// POUs/FileHandling/TF6421-XmlServer/XmlReadWriteWithBackupFile
{attribute 'no_check'}
//Write xml files with a additonal backup file and auto save function if structure will be changed.
//For the Backup functionality, a backup subfolder name "Backup" in the directory is needed! 
//In case the xml could not read successfully after, the backup files will be used.
//See Options to enable auto save and backup file functions.
//based on TF6421 - required lib: Tc2_XmlDataSvr - see Beckhoff documentation for more information
{attribute 'enable_dynamic_creation'}
FUNCTION_BLOCK XmlReadWriteWithBackupFile EXTENDS XmlReadWrite 
VAR_OUTPUT CONSTANT
{attribute 'displaymode':='binary'}
	OPTION_ENABLE_AUTO_SAVE									:	BYTE :=2#0000_0001;
{attribute 'displaymode':='binary'}
	OPTION_ENABLE_BACKUP_FILE								: 	BYTE :=2#0000_0010;
END_VAR                 									
VAR_INPUT               									                       		
{attribute 'displaymode':='binary'}
	Options													:	BYTE := 2#0000_0000;			(* option constants are alreay predefined, so they can accordingly be passed symbolically to the block 
																								Bit 0 = Enable auto save if data changed
																								Bit 1 = Enable backup file 
																								Bit 2 = 
																								Bit 3 = 
																								Bit 4 = 
																								Bit 5 = 
																								Bit 6 = 
																								Bit 7 = 						
																							*)     													
END_VAR
VAR_OUTPUT
	Backup													:	BOOL := FALSE; 		// Backup file has been readed 
	Loaded													:	BOOL:= FALSE;		// Data loaded
	ErrorFnc												:	STRING(30) := ''; 	// Error source
END_VAR
VAR
(* memory ************************************************************)
	rtExecuteAutoSave										:	R_trig;
	pCompareData											:	POINTER TO BYTE;
	pMemSymAddr												: 	PVOID := 0;	
	MemSymSize												:	UDINT;
(* Trigger **********************************************************)

(* timer ******************************************************************)
	tonDelay												:	ton;

(* function blocks ***************************************************************)

(* Dummy **********************************************************)

END_VAR

	(* XML Read/Write with backup file and auto save						V2.2		*)
	(************************************************************************************)

(* reserver memeory for auto save ***************************************************************************************)
	IF Options.0 AND pCompareData = 0 
	THEN	
		pCompareData 										:=  __NEW(BYTE, SymSize);
		IF NOT PARAM.ENABLE_DEBUG_MSG_DYNAMIC_MEM_ALLOCATION
		THEN 
			;
		ELSIF MemSymSize = 0 
		THEN
			AdsLogHint('EngineeringToolbox | FB XmlReadWriteWithBackupFile | An instance allocated %s bytes from the dynamic memory of the ADS router memory pool', TO_STRING(SymSize));	
		ELSE //Allocation of additional memory space
			AdsLogWarn('EngineeringToolbox | FB XmlReadWriteWithBackupFile | An instance allocated additional %s bytes from the dynamic memory of the ADS router memory pool because the size of the data increased (SymSize) ', TO_STRING(SymSize));
		END_IF
		MemSymSize											:= SymSize;
	ELSIF pCompareData <> 0 
	THEN
		IF NOT Options.0 OR SymSize > MemSymSize
		THEN //Delete pointer to allocated memory if no longer needed or size increase 
			__DELETE(pCompareData);
		ELSIF pMemSymAddr <> pSymAddr OR MemSymSize <> SymSize
		THEN //Erease data and rewrite if pointer to data changed or size decreased 
			MEMSET(pCompareData,0,MemSymSize); //Delete compare data if pointer to data changed to activate auto save
			MemSymSize										:= SymSize;
			pMemSymAddr 									:= pSymAddr;	
		END_IF
	END_IF
	
(* Execute sequence ***************************************************************************)	
	rtExecuteAutoSave(CLK := Options.0 AND state = 0 AND Loaded AND pCompareData <> 0 AND_THEN MEMCMP(pSymAddr, pCompareData, SymSize) <> 0);
	rtExecute(CLK := Execute );	
	
	CASE state OF
	0:
		Busy												:= FALSE;
		// init		                                	
		IF NOT Execute                              	
		THEN                                        	
			Backup											:= FALSE;			
			Done 											:= FALSE;
			Error											:= FALSE;
			ErrorID											:= 0;
			ErrorFnc										:= '';
		END_IF                                      	
		                                            	
		IF rtExecute.Q OR rtExecuteAutoSave.Q                       	
		THEN                                        	
			Backup											:= FALSE;
			Done 											:= FALSE;
			Busy											:= TRUE;
			Error											:= FALSE;
			ErrorID											:= 0;
			ErrorFnc										:= '';
			MemFnc											:= SEL(rtExecuteAutoSave.Q, Fnc, FNC_WRITE); // write has priority
			                                        	
			IF pSymAddr = 0                         	
			THEN                                    	
				Busy										:= NOT Error;
				Error										:= TRUE;
				ErrorId										:= E_AdsErr.DEVICE_INVALIDPARM;
				Done										:= FALSE;
				MemFnc										:= -1 ;
				RETURN;                             	
			ELSE
				CASE MemFnc OF
				FNC_READ:	
					XmlSrvRead	(bExecute := FALSE,sFilePath	:= CONCAT(FilePath,FileName));
					state 									:= 10;
				FNC_WRITE:	
					XmlSrvWrite	(bExecute := FALSE,sFilePath	:= CONCAT(FilePath,FileName));
					state 									:= 20;				
				ELSE
					Error									:= TRUE;
					ErrorID									:= E_AdsErr.DEVICE_INVALIDPARM;
					ErrorFnc								:= CONCAT('Invalid Fnc,', INT_TO_STRING(MemFnc));
					Busy									:= FALSE;			
				END_CASE
			END_IF
		END_IF
	
	(* File read ************************************************)
	10:
		XmlSrvRead(                    	
			sNetId		:= NetId,
			ePath		:= ,(* Default *)
			nMode		:= XMLSRV_SKIPMISSING, 
			pSymAddr	:= pSymAddr,
			cbSymSize	:= SymSize,
			sFilePath	:= ,
			sXPath		:= XPath,
			bExecute	:=  TRUE,
			tTimeout	:= Timeout,
			bBusy		=> ,
			bError		=> ,
			nErrId		=> );
			
		IF NOT XmlSrvRead.bBusy
		THEN
			IF XmlSrvRead.bError
			THEN
				IF XmlSrvRead.nErrId = 1804 
					AND Options.1
				THEN
					state									:= 11;
				ELSE
					Error									:= TRUE;
					ErrorID									:= XmlSrvRead.nErrId;
					ErrorFnc								:= CONCAT('XmlSvrRead State:',INT_TO_STRING(State));
					Busy									:= FALSE;
					State									:= 0;	
				END_IF
			ELSE
				Loaded										:= TRUE;
				Busy										:= FALSE;
				Done										:= TRUE;
				MemFnc										:= -1;
				state										:= 0;	
				IF pCompareData <> 0 THEN MEMCPY(pCompareData,pSymAddr,SymSize); pMemSymAddr := pSymAddr; END_IF 	// refresh compare data after reading for initalisation
			END_IF
			XmlSrvRead(bExecute 							:= FALSE);
		END_IF	
				
	11: // Read Backup file
		XmlSrvRead.sFilePath								:= CONCAT(FilePath,'Backup\'); 				// subfolder
		XmlSrvRead.sFilePath								:= CONCAT(XmlSrvRead.sFilePath,FileName);
				
		XmlSrvRead(                    	
			sNetId		:= NetId,
			ePath		:= ,(* Default *)
			nMode		:= XMLSRV_SKIPMISSING, 
			pSymAddr	:= pSymAddr,
			cbSymSize	:= SymSize,
			sFilePath	:= ,
			sXPath		:= XPath,
			bExecute	:=  TRUE,
			tTimeout	:= Timeout,
			bBusy		=> ,
			bError		=> ,
			nErrId		=> );
			
		IF NOT XmlSrvRead.bBusy
		THEN
			IF XmlSrvRead.bError
			THEN
				Error										:= TRUE;
				ErrorID										:= XmlSrvRead.nErrId;
				ErrorFnc									:= CONCAT('XmlSvrRead State:',INT_TO_STRING(State));
				Busy										:= FALSE;
				State										:= 0;	
			ELSE                                        	
				Loaded										:= TRUE;
				Backup										:= TRUE;
				Busy										:= FALSE;
				Done										:= TRUE;
				MemFnc										:= -1;
				state										:= 20; 							// Write original file	
				IF pCompareData <> 0 THEN MEMCPY(pCompareData,pSymAddr,SymSize); pMemSymAddr := pSymAddr; END_IF 	// refresh compare data after reading of backup file for initalisation
			END_IF
			XmlSrvRead(bExecute 							:= FALSE);
		END_IF	
		
	(* Write parameter ***********************************************************)
	20:
		XmlSrvWrite(
			sNetId		:= NetId,
			ePath		:= ,(* Default *)
			nMode		:= Mode,
			pSymAddr	:= pSymAddr,
			cbSymSize	:= SymSize,
			sFilePath	:= ,
			sXPath		:= XPath,
			bExecute	:= TRUE,
			tTimeout	:= Timeout,
			bBusy		=> ,
			bError		=> ,
			nErrId		=> );
			
		IF NOT XmlSrvWrite.bBusy
		THEN
			IF XmlSrvWrite.bError
			THEN
				Error										:= TRUE;
				ErrorID										:= XmlSrvWrite.nErrId;
				ErrorFnc									:= CONCAT('XmlSvrWrite State:',INT_TO_STRING(State));
				Busy										:= FALSE;
				State										:= 0;				
			ELSE // Write backup file	
				Loaded										:= TRUE;
				State										:= SEL(Options.1, 0, 21); //
				Done										:= State = 0; 				
				Busy										:= State <> 0;
				//Update compare memory
				IF pCompareData <> 0 THEN MEMCPY(pCompareData,pSymAddr,SymSize); pMemSymAddr := pSymAddr; END_IF 	// refresh compare data after writing new data
			END_IF
			XmlSrvWrite(bExecute							:= FALSE);
		END_IF

	21://Write backup to sub folder	
		XmlSrvWrite.sFilePath								:= CONCAT(FilePath,'Backup\'); 				// subfolder
		XmlSrvWrite.sFilePath								:= CONCAT(XmlSrvWrite.sFilePath,FileName);
		XmlSrvWrite(
			sNetId		:= NetId,
			ePath		:= ,(* Default *)
			nMode		:= Mode,
			pSymAddr	:= pSymAddr,
			cbSymSize	:= SymSize,
			sFilePath	:= ,
			sXPath		:= XPath,
			bExecute	:= TRUE,
			tTimeout	:= Timeout,
			bBusy		=> ,
			bError		=> ,
			nErrId		=> );
			
		IF NOT XmlSrvWrite.bBusy
		THEN
			IF XmlSrvWrite.bError
			THEN
				Error										:= TRUE;
				ErrorID										:= XmlSrvWrite.nErrId;
				ErrorFnc									:= CONCAT('XmlSvrWrite State:',INT_TO_STRING(State));
				Busy										:= FALSE;
				State										:= 0;				
			ELSE 	
				Busy										:= FALSE;
				Done										:= TRUE;
				State										:= 0;	
				//Update compare memory
				IF pCompareData <> 0 THEN MEMCPY(pCompareData,pSymAddr,SymSize); pMemSymAddr := pSymAddr; END_IF 	// refresh compare data after writing new data				
			END_IF
			XmlSrvWrite(bExecute							:= FALSE);
		END_IF		
	END_CASE
		
		
	
(*************************************************************************************************)

METHOD FB_exit : BOOL
VAR_INPUT
	bInCopyCode : BOOL; // if TRUE, the exit method is called for exiting an instance that is copied afterwards (online change).
END_VAR
IF NOT bInCopyCode AND pCompareData <> 0
THEN //Release memory in case the PLC stopps
	__DELETE(pCompareData);
END_IF
END_METHOD

PROPERTY PUBLIC optEnableAutoSave : BOOL
GET
optEnableAutoSave := Options.0;
END_GET
SET
Options.0 := optEnableAutoSave;
END_SET
END_PROPERTY

PROPERTY PUBLIC optEnableBackupFile : BOOL
GET
optEnableBackupFile := Options.1;
END_GET
SET
Options.1 := optEnableBackupFile;
END_SET
END_PROPERTY

METHOD PUBLIC read : BOOL //Return value = TRUE if busy
//required parameter
//pSymAddr
//SymSize
//FilePath
//XPath
VAR_INPUT
	Execute													:	BOOL;
END_VAR
CASE state OF
0:	
	Fnc 													:= FNC_READ;
	THIS^(Execute:=Execute);
1: 
	;

END_CASE
Read 														:= Busy;
END_METHOD

METHOD PUBLIC write : BOOL //Return value = TRUE if busy
//required parameter
//pSymAddr
//SymSize
//FilePath
//XPath
VAR_INPUT
	Execute													:	BOOL;
END_VAR
CASE state OF
0:	
	Fnc 													:= FNC_WRITE;
	THIS^(Execute:=Execute);
1: 
	;

END_CASE
Write 														:= Busy;
END_METHOD

END_FUNCTION_BLOCK

// POUs/IO/_EcSlaveFWUpdater/EcSlaveDevFWUpdater
FUNCTION_BLOCK EcSlaveDevFWUpdater EXTENDS FbBase
VAR CONSTANT	
	{attribute 'displaymode':='hexadecimal'} 
	COE_FWVERSION_OBJECT								: WORD := 16#100A;
END_VAR
VAR_OUTPUT CONSTANT
	MIN_SLAVE_DEV										:	INT := 1;
	MAX_SLAVE_DEV										:	INT := Param.ETHERCAT_SLAVE_DEV_FW_UPDATER_MAX_DEV;

	{attribute 'displaymode':='binary'}   
	MODE_READ											:	BYTE := 0;
	{attribute 'displaymode':='binary'}   
	MODE_WRITE											:	BYTE := 1;

	{attribute 'displaymode':='binary'}   
	OPTION_WRITE_FW_IF_VERSION_MATCH					:	BYTE := 2#0000_0001;
	
END_VAR
VAR_INPUT
{attribute 'displaymode':='binary'}         			
	Mode												:	BYTE  := 2#0000_0000; 

{attribute 'displaymode':='binary'}  	
	Options												:	BYTE  := 2#0000_0000; 		
				
	PathName											:	STRING; //Path incl. file name of FW file
	RegVersion											:	STRING; //Requested version
	ipSlaveInfoData										:	ARRAY [MIN_SLAVE_DEV..MAX_SLAVE_DEV] OF I_EcSlaveInfoData;
END_VAR
VAR_OUTPUT
	ActVersion											: ARRAY[MIN_SLAVE_DEV..MAX_SLAVE_DEV] OF STRING[20]; 	
	CntFWNOK											: INT; //Count of terminals FW not OK
	TermNo												: INT; //No of terminal in progress
	ProgressWriteFW										: UDINT;	
	VersionRead											: BOOL;
END_VAR
VAR
(*  Memory *****************************************************)
	lastState											: INT := 0;
	MinTerm												: INT;

(*  Timer ******************************************************)
(*  Trigger ****************************************************)

(*  Blocks *****************************************************)
	EcCoeSdoReadEx										: FB_EcCoeSdoReadEx := (nIndex := COE_FWVERSION_OBJECT, tTimeout := DEFAULT_ADS_TIMEOUT);

	CoEFwDownLoad										: FB_EcFoeLoad := (tTimeout := DEFAULT_ADS_TIMEOUT,dwPass := 0, eMode := eFoeMode_Write);
(*  Error ******************************************************)
(*  Dummys *****************************************************)
	{attribute 'hide' := ''}
	i,j													: INT := 0;

END_VAR

	(*********************************************************)
	
(* state machine ********************************************************)
	rtExecute(CLK := Execute);
	CASE state OF
	0 : 
		Busy 											:= FALSE;
		
		IF NOT Execute THEN
			Done 										:= FALSE;
			Error 										:= FALSE;
			ErrorID 									:= 0;
		END_IF
		IF rtExecute.Q THEN
			IF PathName = '' 
			THEN
				Error 									:= TRUE;
				ErrorID 								:= E_AdsErr.DEVICE_INVALIDPARM;

			ELSIF RegVersion = '' AND Mode = MODE_WRITE AND NOT Options.0
			THEN
 				Error 									:= TRUE;
				ErrorID 								:= E_AdsErr.DEVICE_INVALIDPARM; 
									
			ELSIF ipSlaveInfoData[MIN_SLAVE_DEV] = 0
			THEN
 				Error 									:= TRUE;
				ErrorID 								:= E_AdsErr.DEVICE_INVALIDPARM; 			
			ELSE
				Busy									:= TRUE;	
				Done 									:= FALSE;
				Error 									:= FALSE;
				ErrorID 								:= 0;
				TermNo									:= MIN_SLAVE_DEV;	
				ProgressWriteFW							:= 0;
				CntFWNOK								:= 0;					
				
			
				EcCoeSdoReadEx(bExecute := FALSE);
				CoEFwDownLoad(bExecute := FALSE);
				state									:= SEL(Mode = MODE_READ, 1, 2);
			END_IF
		END_IF
			
	1: (* Write FW *****************************************************************)
		CoEFwDownLoad(
			bExecute		:= ipSlaveInfoData[TermNo].rInfoData.AdsAddr.port <> 0 AND (ActVersion[TermNo] <> RegVersion OR Options.0) , 
			sNetId			:= F_CreateAmsNetId(nIds := ipSlaveInfoData[TermNo].rInfoData.AdsAddr.netId),
			nSlaveAddr		:= ipSlaveInfoData[TermNo].rInfoData.AdsAddr.port,
			sPathName		:= PathName,
			nProgress 		=> ProgressWriteFW);	
		IF NOT 	CoEFwDownLoad.bBusy
		THEN
			ProgressWriteFW								:= 0;
			IF CoEFwDownLoad.bError
			THEN
				ErrorID									:= EcCoESdoReadEx.nErrId;
				CntFWNOK								:= CntFWNOK + 1;	
				ActVersion[TermNo]						:= 'ERR_DOWNLOADING';
			ELSIF CoEFwDownLoad.bExecute	
			THEN
				ActVersion[TermNo]						:= 'DOWNLOADED';
			ELSE
				ActVersion[TermNo]						:= '------';
			END_IF
			//Next terminal
			TermNo										:= TermNo + 1;
			
			IF TermNo > MAX_SLAVE_DEV 
				OR ipSlaveInfoData[TermNo] = 0
			THEN //Start reading
				MEMSET(ADR(ActVersion),0,SIZEOF(ActVersion));
				VersionRead								:= FALSE;
				TermNo									:= MIN_SLAVE_DEV;		
				state									:= 2;
			END_IF		
			CoEFwDownLoad(bExecute := FALSE);
		ELSE
			ActVersion[TermNo]							:= CONCAT('DOWNLOADING ',CONCAT(TO_STRING(CoEFwDownLoad.nProgress),'%'));
		END_IF
	
	2: (* Read FW Version **********************************************************)
		EcCoESdoReadEx(
			bExecute		:= ipSlaveInfoData[TermNo].rInfoData.AdsAddr.port <> 0,
			sNetId			:= F_CreateAmsNetId(nIds := ipSlaveInfoData[TermNo].rInfoData.AdsAddr.netId),
			nSlaveAddr		:= ipSlaveInfoData[TermNo].rInfoData.AdsAddr.port,
			pDstBuf			:= ADR(ActVersion[TermNo]),
			cbBufLen		:= SIZEOF(ActVersion[TermNo]));
		IF NOT EcCoESdoReadEx.bBusy
		THEN
			IF EcCoESdoReadEx.bError 
			THEN
				ActVersion[TermNo]						:= 'ERR_READING';
				ErrorID									:= EcCoESdoReadEx.nErrId;
				CntFWNOK								:= CntFWNOK + 1;	
			ELSIF NOT EcCoESdoReadEx.bExecute 
			THEN
				ActVersion[TermNo]						:= 'NOT_CONNECTED';
			ELSIF ActVersion[TermNo] <> RegVersion
			THEN
				CntFWNOK								:= CntFWNOK + 1;	
			END_IF
			
			//Next terminal
			TermNo										:= TermNo + 1;
			
			IF TermNo > MAX_SLAVE_DEV
				OR ipSlaveInfoData[TermNo] = 0
			THEN
				TermNo									:= MAX_SLAVE_DEV;
				Done									:= CntFWNOK = 0;
				VersionRead								:= TRUE;
				Error									:= NOT Done;
				Busy									:= FALSE;
				state									:= 0;
			END_IF
			EcCoeSdoReadEx(bExecute := FALSE);
		END_IF
	END_CASE	

(* Record last state ******************************************)
IF state <> lastState AND state <> 0 AND NOT Error
THEN 
	lastState											:= state;
END_IF

(*************************************************************)

END_FUNCTION_BLOCK

// POUs/IO/_ItfActuators/I_ActuatorBase
INTERFACE I_ActuatorBase EXTENDS __System.IQueryInterface

{attribute 'monitoring' := 'call'}
PROPERTY public inError : bool
GET
END_GET
END_PROPERTY

{attribute 'monitoring' := 'call'}
PROPERTY public isBusy : bool
GET
END_GET
END_PROPERTY

{attribute 'monitoring' := 'call'}
PROPERTY public isOff : BOOL
GET
END_GET
END_PROPERTY

{attribute 'monitoring' := 'call'}
PROPERTY public noFeed : BOOL
GET
END_GET
END_PROPERTY

{attribute 'monitoring' := 'call'}
PROPERTY public ok : bool
GET
END_GET
END_PROPERTY

METHOD PUBLIC reset : BOOL
VAR_INPUT
END_VAR
END_METHOD

METHOD public switchOff : BOOL
VAR_INPUT
END_VAR
END_METHOD

END_INTERFACE

// POUs/IO/_ItfActuators/I_ActuatorEnableDisable
INTERFACE I_ActuatorEnableDisable EXTENDS I_ActuatorBase

{attribute 'monitoring' := 'call'}
PROPERTY public isDisabled : BOOL
GET
END_GET
END_PROPERTY

{attribute 'monitoring' := 'call'}
PROPERTY public isEnabled : BOOL
GET
END_GET
END_PROPERTY

METHOD public setDisable : BOOL
VAR_INPUT
END_VAR
END_METHOD

METHOD public setEnable : BOOL
VAR_INPUT
END_VAR
END_METHOD

END_INTERFACE

// POUs/IO/_ItfActuators/I_ActuatorFwdBwd
INTERFACE I_ActuatorFwdBwd EXTENDS I_ActuatorBase

{attribute 'monitoring' := 'call'}
PROPERTY public backwardStarted : BOOL
GET
END_GET
END_PROPERTY

{attribute 'monitoring' := 'call'}
PROPERTY public forwardStarted : BOOL
GET
END_GET
END_PROPERTY

METHOD public startBackward : BOOL
VAR_INPUT
END_VAR
END_METHOD

METHOD public startForward : BOOL
VAR_INPUT
END_VAR
END_METHOD

END_INTERFACE

// POUs/IO/_ItfActuators/I_ActuatorFwdRev
INTERFACE I_ActuatorFwdRev EXTENDS I_ActuatorBase

{attribute 'monitoring' := 'call'}
PROPERTY public forwardStarted : BOOL
GET
END_GET
END_PROPERTY

{attribute 'monitoring' := 'call'}
PROPERTY public reverseStarted : BOOL
GET
END_GET
END_PROPERTY

METHOD public startForward : BOOL
VAR_INPUT
END_VAR
END_METHOD

METHOD public startReverse : BOOL
VAR_INPUT
END_VAR
END_METHOD

END_INTERFACE

// POUs/IO/_ItfActuators/I_ActuatorLeftRight
INTERFACE I_ActuatorLeftRight EXTENDS I_ActuatorBase

{attribute 'monitoring' := 'call'}
PROPERTY public leftOk : BOOL
GET
END_GET
END_PROPERTY

{attribute 'monitoring' := 'call'}
PROPERTY public rightOk : BOOL
GET
END_GET
END_PROPERTY

METHOD public toTheLeft : BOOL
VAR_INPUT
END_VAR
END_METHOD

METHOD public toTheRight : BOOL
VAR_INPUT
END_VAR
END_METHOD

END_INTERFACE

// POUs/IO/_ItfActuators/I_ActuatorOnOff
INTERFACE I_ActuatorOnOff EXTENDS I_ActuatorBase

{attribute 'monitoring' := 'call'}
PROPERTY public isOn : BOOL
GET
END_GET
END_PROPERTY

METHOD public switchOn : BOOL
VAR_INPUT
END_VAR
END_METHOD

END_INTERFACE

// POUs/IO/_ItfActuators/I_ActuatorOpenClose
INTERFACE I_ActuatorOpenClose EXTENDS I_ActuatorBase

{attribute 'monitoring' := 'call'}
PROPERTY public isClosed : BOOL
GET
END_GET
END_PROPERTY

{attribute 'monitoring' := 'call'}
PROPERTY public isOpened : BOOL
GET
END_GET
END_PROPERTY

METHOD public setClose : BOOL
VAR_INPUT
END_VAR
END_METHOD

METHOD public setOpen : BOOL
VAR_INPUT
END_VAR
END_METHOD

END_INTERFACE

// POUs/IO/_ItfActuators/I_ActuatorPosNeg
INTERFACE I_ActuatorPosNeg EXTENDS I_ActuatorBase

{attribute 'monitoring' := 'call'}
PROPERTY public negativeOk : BOOL
GET
END_GET
END_PROPERTY

METHOD PUBLIC negativeOn : BOOL
VAR_INPUT
END_VAR
END_METHOD

{attribute 'monitoring' := 'call'}
PROPERTY public positiveOk : BOOL
GET
END_GET
END_PROPERTY

METHOD PUBLIC positiveOn : BOOL
VAR_INPUT
END_VAR
END_METHOD

END_INTERFACE

// POUs/IO/_ItfActuators/I_ActuatorStartStop
INTERFACE I_ActuatorStartStop EXTENDS I_ActuatorBase

{attribute 'monitoring' := 'call'}
PROPERTY public isStarted : BOOL
GET
END_GET
END_PROPERTY

{attribute 'monitoring' := 'call'}
PROPERTY public isStopped : BOOL
GET
END_GET
END_PROPERTY

METHOD public start : BOOL
VAR_INPUT
END_VAR
END_METHOD

METHOD public stop : BOOL
VAR_INPUT
END_VAR
END_METHOD

END_INTERFACE

// POUs/IO/_ItfActuators/I_ActuatorUpDown
INTERFACE I_ActuatorUpDown EXTENDS I_ActuatorBase

{attribute 'monitoring' := 'call'}
PROPERTY public downOk : BOOL
GET
END_GET
END_PROPERTY

METHOD public moveDown : BOOL
VAR_INPUT
END_VAR
END_METHOD

METHOD public moveUp : BOOL
VAR_INPUT
END_VAR
END_METHOD

{attribute 'monitoring' := 'call'}
PROPERTY public upOK : BOOL
GET
END_GET
END_PROPERTY

END_INTERFACE

// POUs/IO/_ItfActuators/I_ActuatorWorkBase
INTERFACE I_ActuatorWorkBase EXTENDS I_ActuatorBase

{attribute 'monitoring' := 'call'}
PROPERTY isInBasePos : BOOL
GET
END_GET
END_PROPERTY

{attribute 'monitoring' := 'call'}
PROPERTY isInWorkPos : BOOL
GET
END_GET
END_PROPERTY

METHOD public moveToBasePos : BOOL
VAR_INPUT
END_VAR
END_METHOD

METHOD public moveToWorkPos : BOOL
VAR_INPUT
END_VAR
END_METHOD

END_INTERFACE

// POUs/IO/Analog/AnalogIn32
{attribute 'no_check'}
FUNCTION_BLOCK AnalogIn32 extends EcSlaveInfoDataExt
VAR_INPUT
	MinValue												: 	LREAL 	:= 0.0;
	MaxValue												: 	LREAL 	:= 0.0;
	NoOfDigits												: 	INT 	(0..10)	:= 0; //number of decimal digits of scaled Q variable 
	OutOnError												:	LREAL 	:= 0.000000000000000001;
{attribute 'displaymode':='binary'}     	            	
	Options													:	BYTE  := 2#0000_0010; (* .0 = FALSE Scale value from 0 to e.g. 32767 / TRUE scale singed value e.g. -32768 <-> 32767 , see Options .1 and .2 for more scaling Options 
																						.1 = FALSE = 32 bit resolution / TRUE = value is based on 24 bit resolution e.g. -> -8388608.0 or 0.0 <-> 8388607.0 
																						.2 = Right adjust of 32/24 bit value -> value will be shifted by 8 bits (divided bv 256)   
																						.3 = TRUE = Enable extended range mode -> change scaling to +/-7812500 instead of r+/- 838860x *)
	Offset													:	LREAL := 0.0;
END_VAR                 									                                	            	
VAR_OUTPUT                              	            	
	Q														:	LREAL;	//scaled result value
	In											AT  %I* 	: 	DINT; 	//Hardware Input 
{attribute 'displaymode':='binary'}     	            	
	Status										AT  %I*		:	WORD := 2#0100_0000_0000_0000;	//Terminal status word -> can also be linked with status byte
END_VAR

(* read 32bit analog value 																				    *)
(* resolution process image			e.g.				/ 0V = 0 / 10V = 2147483647 / -10V = - 2147483647 	*)
(* or directly with NoOfDigits																	250 -> 25.0°*)
(************************************************************************************************************)
	
(* Scaling ******************************************************************)
	IF MaxValue <> MinValue 
	THEN
		IF Options.1 
		THEN //24 bit resolution
			IF NOT Options.3
			THEN
				Q 	 										:= Offset + scale(SEL(Options.2 , In , In / 256.0 ) , SEL(Options.0, 0.0, -8388608.0), 8388607.0, MinValue , MaxValue);
			ELSE
		 		Q 	 										:= Offset + scale(SEL(Options.2 , In , In / 256.0 ) , SEL(Options.0, 0.0, -7812500.0), 7812500.0, MinValue , MaxValue);
			END_IF
		ELSE //32 bit resolution 
			Q 	 											:= Offset + scale(SEL(Options.2 , In , In / 256.0 ) , SEL(Options.0, 0.0, -2147483648.0), 2147483647.0, MinValue , MaxValue);		
		END_IF
		IF NoOfDigits > 0
		THEN
			Q												:= TO_FMLREAL(Q,NoOfDigits);
		END_IF
	
	ELSIF NoOfDigits > 0 (* Bsp PT100 *)
	THEN
		Q													:= Offset + TO_FMLREAL(In,NoOfDigits);
		
	ELSE  													
		Q 													:= 0.0;
	END_IF

	IF 	Error AND OutOnError <> 0.000000000000000001
	THEN
		Q													:= OutOnError;
	END_IF
(**********************************************************************************************************************)

{attribute 'monitoring' := 'call'}
PROPERTY PUBLIC Error : BOOL
GET
Error					:= Status.6 OR MinValue = MaxValue AND NoOfDigits = 0;
END_GET
END_PROPERTY

{attribute 'monitoring' := 'call'}
PROPERTY PUBLIC Limit_1 : BYTE
GET
Limit_1.0					:= Status.2;
Limit_1.1					:= Status.3;
END_GET
END_PROPERTY

{attribute 'monitoring' := 'call'}
PROPERTY PUBLIC Limit_2 : BYTE
GET
Limit_2.0					:= Status.4;
Limit_2.1					:= Status.5;
END_GET
END_PROPERTY

PROPERTY optEnable24BitResolution : BOOL //In value is provided as 32bit value instead if 24bit
GET
optEnable24BitResolution := Options.1;
END_GET
SET
Options.1 := optEnable24BitResolution;
END_SET
END_PROPERTY

PROPERTY PUBLIC optEnableScaleExtRangeMode : bool
GET
optEnableScaleExtRangeMode := Options.3;
END_GET
SET
Options.3 := optEnableScaleExtRangeMode;
END_SET
END_PROPERTY

PROPERTY PUBLIC optEnableScaleSignedValue : bool
GET
optEnableScaleSignedValue := Options.0;
END_GET
SET
Options.0 := optEnableScaleSignedValue;
END_SET
END_PROPERTY

PROPERTY PUBLIC optShiftValueBy8Bits : BOOL
GET
optShiftValueBy8Bits := Options.2;
END_GET
SET
Options.2 := optShiftValueBy8Bits;
END_SET
END_PROPERTY

{attribute 'monitoring' := 'call'}
PROPERTY PUBLIC Overrange : BOOL
GET
Overrange					:= Status.1;
END_GET
END_PROPERTY

{attribute 'monitoring' := 'call'}
PROPERTY PUBLIC SyncError : BOOL
GET
SyncError 			:= Status.13;
END_GET
END_PROPERTY

{attribute 'monitoring' := 'call'}
PROPERTY PUBLIC TxPDOState : BOOL
GET
TxPDOState					:= Status.14; //True if not valid
END_GET
END_PROPERTY

{attribute 'monitoring' := 'call'}
PROPERTY PUBLIC TxPDOToggle : BOOL
GET
TxPDOToggle						:= Status.15;
END_GET
END_PROPERTY

{attribute 'monitoring' := 'call'}
PROPERTY PUBLIC Underrange : BOOL
GET
Underrange 					:= Status.0;
END_GET
END_PROPERTY

END_FUNCTION_BLOCK

// POUs/IO/Analog/AnalogInELMBase
// Based FB for analog input channels of ELM terminals incl. EtherCAT Slave Info Data 
//You can inherit your final implementation from this base "class"  
FUNCTION_BLOCK AnalogInELMBase EXTENDS EcSlaveInfoData
VAR_INPUT
	Enable													:	BOOL 	:= TRUE;
	MinValue												: 	LREAL 	:= 0.0;
	MaxValue												: 	LREAL 	:= 0.0;
	NoOfDigits												: 	INT 	(0..10)	:= 0; //number of decimal digits of scaled Q variable 
	OutOnError												:	LREAL 	:= 0.000000000000000001;
{attribute 'displaymode':='binary'}     	            	
	Options													:	BYTE  := 2#0000_0000;
END_VAR                 									
VAR                                     	            	
{attribute 'displaymode':='binary'}     	            	
	Status										AT  %I*		:	DWORD := 2#0100_0000_0000_0000;	//Terminal status (4 bytes) 
	
END_VAR                                 	            	
VAR_OUTPUT                              	            	                                       	
	(* Statusbist *)                    	
	NoOfSamples												:	USINT; //Byte 1
	Error													:	BOOL; //Byte2.0
	Underrange 												:	BOOL; //Byte2.1
	Overrange												:	BOOL ; //Byte2.2
	Diag													:	BOOL; //Byte2.4
	TxPDOState												:	BOOL; //Byte2.5
	InputCycleCounter										:	USINT; //Byte2.6/.7	
END_VAR                                 	
VAR                                     	
END_VAR

(* Base FB for ELM analog in terminals 																		*)
(************************************************************************************************************)

(* evaluate statusword **************************************************************************************)
	MEMCPY(ADR(NoOfSamples),ADR(Status),SIZEOF(NoOfSamples));
	Error													:= Enable AND (Status.8 OR MinValue = MaxValue AND NoOfDigits = 0);
	Underrange 												:= Status.9;
	Overrange												:= Status.10;
	
	Diag													:= Status.12;
	TxPDOState												:= Status.13; //True if not valid
	InputCycleCounter.0										:= Status.14;
	InputCycleCounter.1										:= Status.15;
	
(**********************************************************************************************************************)

END_FUNCTION_BLOCK

// POUs/IO/Analog/AnalogInELMSingleSampleDINT
// AnalogIn FB to read and scale a single DINT (24bit) sample input from ELMxxxx terminal
// Set bit 3 (Options.3) to true to enable scaling based on +/-7812500 instead of legacy range values +/-838860x
FUNCTION_BLOCK AnalogInELMSingleSampleDINT EXTENDS AnalogInELMBase
VAR_INPUT
	Offset													:	LREAL := 0.0;

END_VAR                 									
VAR                                     	            	
END_VAR                                 	            	
VAR_OUTPUT                              	            	                                       	
	Q														:	LREAL;	//scaled result value
	In											AT  %I* 	: 	DINT; 	//Hardware Input 
END_VAR                                 	
VAR                                   	
END_VAR

(* Read single DINT sample value from ELM terminal and scale to user units									*)
(************************************************************************************************************)

(* evaluate statusword **************************************************************************************)
	SUPER^();
	
(* Scaling ******************************************************************)
	IF MaxValue <> MinValue 
	THEN	
		IF NOT Options.3
		THEN
			Q 	 											:= Offset + Scale(TO_LREAL(In) , -8388608.0, 8388607.0, MinValue , MaxValue);
		ELSE
			Q 	 											:= Offset + Scale(TO_LREAL(In), -7812500.0, 7812500.0, MinValue , MaxValue);
		END_IF	
		IF NoOfDigits > 0
		THEN
			Q												:= TO_FMLREAL(Q,NoOfDigits);
		END_IF
	
	ELSIF NoOfDigits > 0 (* Bsp PT100 *)
	THEN
		Q													:= Offset + TO_FMLREAL(In,NoOfDigits);
		
	ELSE  													
		Q 													:= 0.0;
	END_IF

	IF 	Error AND OutOnError <> 0.000000000000000001
	THEN
		Q													:= OutOnError;
	END_IF
(**********************************************************************************************************************)

METHOD FB_init : BOOL
VAR_INPUT
	bInitRetains : BOOL; // if TRUE, the retain variables are initialized (warm start / cold start)
	bInCopyCode : BOOL;  // if TRUE, the instance afterwards gets moved into the copy code (online change)
END_VAR
IF NOT bInCopyCode THEN
	NoOfDigits 							:= 2;
END_IF
END_METHOD

PROPERTY PUBLIC optEnableScaleExtRangeMode : bool
GET
optEnableScaleExtRangeMode := Options.3;
END_GET
SET
Options.3 := optEnableScaleExtRangeMode;
END_SET
END_PROPERTY

END_FUNCTION_BLOCK

// POUs/IO/Analog/AnalogInELMSingleSampleREAL
// AnalogIn FB to read and scale a single REAL sample input from ELMxxxx terminal
// Set bit 3 (Options.3) to true to enable scaling based on +/-7812500 instead of legacy range values +/-838860x
// NoOfDigits per default set to 3... 
FUNCTION_BLOCK AnalogInELMSingleSampleREAL EXTENDS AnalogInELMBase
VAR_INPUT
	Offset													:	LREAL := 0.0;
END_VAR                 									
VAR                                     	            	
END_VAR                                 	            	
VAR_OUTPUT                              	            	                                       	
	Q														:	LREAL;	//scaled result value
	In											AT  %I* 	: 	REAL; 	//Hardware Input 
END_VAR                                 	
VAR                                     	
END_VAR

(* Read single REAL sample value from ELM terminal and scale to user units									*)
(************************************************************************************************************)

(* evaluate statusword **************************************************************************************)
	SUPER^();
	
(* Scaling ******************************************************************)
	IF MaxValue <> MinValue 
	THEN			
		IF NOT Options.3
		THEN
			Q 	 											:= Offset + Scale(TO_LREAL(In), -8388608.0, 8388607.0, MinValue , MaxValue);
		ELSE
			Q 	 											:= Offset + Scale(TO_LREAL(In),  -7812500.0, 7812500.0, MinValue , MaxValue);		
		END_IF	
		
		IF NoOfDigits > 0
		THEN
			Q												:= TO_FMLREAL(Q,NoOfDigits);
		END_IF
	
	ELSIF NoOfDigits > 0 (* Bsp PT100 *)
	THEN
		Q													:= Offset + TO_FMLREAL(In,NoOfDigits);
		
	ELSE  													
		Q 													:= 0.0;
	END_IF


(**********************************************************************************************************************)

METHOD FB_init : BOOL
VAR_INPUT
	bInitRetains : BOOL; // if TRUE, the retain variables are initialized (warm start / cold start)
	bInCopyCode : BOOL;  // if TRUE, the instance afterwards gets moved into the copy code (online change)
END_VAR
IF NOT bInCopyCode THEN
	NoOfDigits 							:= 3;
END_IF
END_METHOD

PROPERTY PUBLIC optEnableScaleExtRangeMode : bool
GET
optEnableScaleExtRangeMode := Options.3;
END_GET
SET
Options.3 := optEnableScaleExtRangeMode;
END_SET
END_PROPERTY

END_FUNCTION_BLOCK

// POUs/IO/Analog/AnalogInREAL
// AnalogInReal FB to read and scale a single REAL input
// Set bit 3 (Options.3) to true to enable scaling based on +/-7812500 instead of legacy range values +/-838860x
// NoOfDigits per default set to 3... 
FUNCTION_BLOCK AnalogInREAL EXTENDS EcSlaveInfoDataExt
VAR_INPUT
	Offset													:	LREAL 		:= 0.0;
	MinValue												: 	LREAL 		:= 0.0;
	MaxValue												: 	LREAL 		:= 0.0;
	NoOfDigits												: 	INT(0..10)	:= 0; //number of decimal digits of scaled Q variable 
	OutOnError												:	LREAL 		:= 0.000000000000000001;
{attribute 'displaymode':='binary'}     	            	
	Options													:	BYTE  		:= 2#0000_0000;
END_VAR                 									
VAR                        
END_VAR                                 	            	
VAR_OUTPUT                              	            	                                       	
	Q														:	LREAL;//scaled result value
	In											AT  %I* 	: 	REAL; //Hardware Input
	{attribute 'displaymode':='binary'}     	            	
	Status										AT  %I*		:	WORD := 2#00000000_00000000;	//Terminal status (2 bytes)
END_VAR

(* Read single REAL value from terminal and scale to user units				*)
(****************************************************************************)

(* Scaling ******************************************************************)
	IF MaxValue <> MinValue 
	THEN			
		IF NOT Options.3
		THEN
			Q 	 											:= Offset + Scale(TO_LREAL(In), -8388608.0, 8388607.0, MinValue , MaxValue);
		ELSE
			Q 	 											:= Offset + Scale(TO_LREAL(In),  -7812500.0, 7812500.0, MinValue , MaxValue);		
		END_IF	
		
		IF NoOfDigits > 0
		THEN
			Q												:= TO_FMLREAL(Q,NoOfDigits);
		END_IF
	
	ELSIF NoOfDigits > 0 (* Bsp PT100 *)
	THEN
		Q													:= Offset + TO_FMLREAL(In,NoOfDigits);
		
	ELSE  													
		Q 													:= 0.0;
	END_IF

(****************************************************************************)

{attribute 'monitoring' := 'call'}
PROPERTY PUBLIC Error : BOOL
GET
Error					:= Status.6 OR MinValue = MaxValue AND NoOfDigits = 0;
END_GET
END_PROPERTY

{attribute 'monitoring' := 'call'}
PROPERTY PUBLIC Limit_1 : BYTE
GET
Limit_1.0					:= Status.2;
Limit_1.1					:= Status.3;
END_GET
END_PROPERTY

{attribute 'monitoring' := 'call'}
PROPERTY PUBLIC Limit_2 : BYTE
GET
Limit_2.0					:= Status.4;
Limit_2.1					:= Status.5;
END_GET
END_PROPERTY

PROPERTY PUBLIC optEnableScaleExtRangeMode : bool
GET
optEnableScaleExtRangeMode := Options.3;
END_GET
SET
Options.3 := optEnableScaleExtRangeMode;
END_SET
END_PROPERTY

{attribute 'monitoring' := 'call'}
PROPERTY PUBLIC Overrange : BOOL
GET
Overrange 			:= Status.1;
END_GET
END_PROPERTY

{attribute 'monitoring' := 'call'}
PROPERTY PUBLIC TareActive : BOOL
GET
TareActive					:= Status.11;
END_GET
END_PROPERTY

{attribute 'monitoring' := 'call'}
PROPERTY PUBLIC TxPDOState : BOOL
GET
TxPDOState					:= Status.14; //True if not valid
END_GET
END_PROPERTY

{attribute 'monitoring' := 'call'}
PROPERTY PUBLIC TxPDOToggle : BOOL
GET
TxPDOToggle							:= Status.15;
END_GET
END_PROPERTY

{attribute 'monitoring' := 'call'}
PROPERTY PUBLIC Underrange : BOOL
GET
Underrange 			:= Status.0;
END_GET
END_PROPERTY

END_FUNCTION_BLOCK

// POUs/IO/Analog/AnalogOut
{attribute 'no_check'}
//Provides an INT output varibale (Q	AT  %Q* : 	INT) to writed a scaled lreal value to an anallog output (terminal)
FUNCTION_BLOCK AnalogOut
VAR_INPUT
	SetValue												: 	LREAL 	:= 0.0;	
	MinValue												: 	LREAL 	:= 0.0;
	MaxValue												: 	LREAL 	:= 0.0;	
{attribute 'displaymode':='binary'}
	Options													:	BYTE 	:= 2#0000_0000; (* .0 = FALSE scale output to 0 - 32767 / TRUE = scale output from -32768 to +32767 *)
END_VAR             							
VAR_OUTPUT          							
	Q												AT  %Q* : 	INT; (* Hardware Output *)
END_VAR             							
VAR                 							
	x														:	LREAL;
END_VAR

(* Analogvalue output	 													    *)
(* resolution  							/ 0V = 0 / 10V = 32768 / -10V = - 32767 *)
(********************************************************************************)

(* standardization **************************************************************)
	Q															:= TO_INT(Scale(SetValue,MinValue,MAxValue,SEL(Options.0 , 0.0  , -32768.0), 32767.0));		

(*********************************************************************************)

PROPERTY PUBLIC optEnableScaleSignedValue : bool
GET
optEnableScaleSignedValue := Options.0;
END_GET
SET
Options.0 := optEnableScaleSignedValue;
END_SET
END_PROPERTY

END_FUNCTION_BLOCK

// POUs/IO/Cylinder/Cylinder
{attribute 'no_check'}
//Cylinder object with two outputs (Workpos./Basepos) and correlated inputs
//Via the Options byte, it is possible to disable the use either of one or both feedback inputs.
//In case the physical feedback input in disabled, the status output of the FB will be generated by PT_Feedback
//In case the physical feedback input will not be triggerd to his corresonding outout within a certain time (PT_Feedback), an timeout error occures
//The physical outputs could be blocked by set the FeedxxxPos signals to false.
//FB "INPUT" is used inside
FUNCTION_BLOCK Cylinder IMPLEMENTS I_Cylinder
VAR_OUTPUT CONSTANT
{attribute 'displaymode':='binary'}
	OPTION_DISABLE_SENSOR_BASEPOS							:	BYTE  := 2#0000_0001; //Disable sensor check basepos. Feedback time used instead to create signal
{attribute 'displaymode':='binary'}
	OPTION_DISABLE_SENSOR_WORKPOS							:	BYTE  := 2#0000_0010; //Disable sensor check workpos. Feedback time used instead to create signal
{attribute 'displaymode':='binary'}
	OPTION_FREE												:	BYTE  := 2#0000_0100; //Not used option		
{attribute 'displaymode':='binary'}
	OPTION_DISABLE_LOGIC_ERROR								:	BYTE  := 2#0000_1000; //Disable logic error (Sensor workpos and basepos active at the same time) 	
{attribute 'displaymode':='binary'}
	OPTION_SWAP_SENSOR_STATUS								:	BYTE  := 2#0001_0000; //Swap signals work and base pos at Status byte
{attribute 'displaymode':='binary'}
	OPTION_INVERT_SENSOR_BASEPOS							:	BYTE  := 2#0010_0000; //Invert logic of sensor basepos (->NO)
{attribute 'displaymode':='binary'}
	OPTION_INVERT_SENSOR_WORKPOS							:	BYTE  := 2#0100_0000;//Invert logic of sensor workpos (->NO)
{attribute 'displaymode':='binary'}
	OPTION_EN_IMPULS_VALVE									:	BYTE  := 2#1000_0000; //Outputs are switched off if endposition is reached	
END_VAR
VAR_INPUT  (* Peripherie Outputs *)
	Quit													:	BOOL;	//Resets error with rising edge
	ToWorkPos												:	BOOL;	//moves cylinder to work position
	ToBasePos												:	BOOL;	//moves cylinder to base position
{attribute 'displaymode':='binary'}         			
	Options													:	BYTE  := 2#0000_0000;  (* option constants are predefined, so they can accordingly be passed symbolically to the block
																							DISABLE_FEEDBACK_BP	= .0
																							DISABLE_FEEDBACK_WP	= .1
																							ENABLE_LATCH_ERROR	= .2
																							DISABLE_LOGIC_ERROR	= .3																							
																							SWAP_SENSOR_STATUS	= .4
																							FEEDBACK_BP_INVERT	= .5
																							FEEDBACK_WP_INVERT	= .6
																							IMPULS_VALVE		= .7
																									*)
	FeedBasePos												:	BOOL := TRUE;	//enables feed in base direction
	FeedWorkPos												:	BOOL := TRUE;	//enables feed in work direction
	PT_Timeout												:	TIME := T#5S; 	//Runtime check BasePos
	PT_Feedback												:	TIME := T#3S; 	//Delay simulate Feedback
	PT_SensorDamping										:	TIME := T#0MS; 	//Work and Base pos sensor on/off damping time to suppress sensor flickering  
END_VAR                                     			
VAR_OUTPUT  (* Peripherie Inputs *)         			
	InBasePos												:	BOOL;	//TRUE when cylinder is in base position
	InWorkPos												:	BOOL;	//TRUE when cylinder is in work position
	Done													:	BOOL; 	//Limit sensor reached or feedback time counted down
	Busy													:	BOOL;	//Busy is TRUE at the rising edge of Execute and FALSE when one of the outputs Done, Aborted, or Error is set 
	ErrBasePos												:	BOOL;	//Cannot reach base position
	ErrWorkPos												:	BOOL;	//Cannot reach work position  
	ErrLogic												:	BOOL; 	//Both feedback signals are on
{attribute 'displaymode':='binary'}         			
	Status													:	BYTE;	(* 	Bit 0 = Q_ToBasePos or opposite if status swap in Options is active
																			Bit 1 = Q_ToWorkPos or opposite if status swap in Options is active
																			Bit 2 = InBasePos or opposite if status swap in Options is active
																			Bit 3 = InWorkPos or opposite if status swap in Options is active
																			Bit 4 = FeedBasePos or opposite if status swap in Options is active
																			Bit 5 = FeedWorkPos or opposite if status swap in Options is active
																			Bit 6 = Ready (no error)
																			Bit 7 = Error timeout move to position or sensor logic
																		*)
	Q_ToBasePos										AT  %Q* :	BOOL; //Hardware output - only with read access
	Q_ToWorkPos										AT  %Q* :	BOOL; //Hardware output - only with read access
END_VAR
VAR// IOs 
	SensorBasePos											: INPUT;
	SensorWorkPos											: INPUT;	
	TonErrBasePos											: TON;
	TonErrWorkPos											: TON;
	SimulationOn											:	BOOL;
END_VAR

	(* Cylinder	 IO V2.9					 								       	*)
	(* Includes functionblock "INPUT" 												*)
	(********************************************************************************)

(* Write Output *****************************************************)
	IF ToBasePos 	
	THEN
		moveToBasePos();
	ELSIF ToWorkPos AND NOT ToBasePos
	THEN
		moveToWorkPos();
	ELSE
		switchOff();
	END_IF

(* Reedkontakte lesen ***********************************************)
	this^._readSensors();
	
(* Status *************************************************)
	_writeStatus();
                        	
(* ack Error **********************************************************)
	IF Quit  THEN  reset(); END_IF

(* Timeout  ************************************************)
	_runtimeChk();
	
(*********************************************************************)

METHOD PROTECTED _readSensors : BOOL
VAR_INPUT
END_VAR
	SensorBasePos(
		Force	:= Q_ToBasePos AND NOT InWorkPos AND(Options.0 OR SimulationOn),
		Invert	:= Options.5,
		PT_ON	:= SEL(Options.0 OR SimulationOn,PT_SensorDamping,PT_FEEDBACK),
		PT_OFF	:= SEL(Options.0 OR SimulationOn,PT_SensorDamping,T#0MS),
		Q_DIRECT=>,
		Q		=> InBasePos,
		Q_RT	=> ,
		Q_FT	=> ,
		IN		=> );


	SensorWorkPos(
		Force	:= Q_ToWorkPos AND NOT InBasePos AND(Options.1 OR SimulationOn),
		Invert	:= Options.6,
		PT_ON	:= SEL(Options.1 OR SimulationOn ,PT_SensorDamping,PT_FEEDBACK),
		PT_OFF	:= SEL(Options.1 OR SimulationOn ,PT_SensorDamping,T#0MS),
		Q_DIRECT=>,
		Q		=> InWorkPos,
		Q_RT	=> ,
		Q_FT	=> ,
		IN		=> );
		

	_readSensors									:= TRUE;
END_METHOD

METHOD PROTECTED _runtimeChk : BOOL
VAR_INPUT
END_VAR
(* Timeout WorkPos ************************************************)
	TonErrWorkPos(	IN := Q_ToWorkPos AND (NOT InWorkPos OR InBasePos),
					PT := MAX(PT_Timeout + PT_SensorDamping,PT_Feedback + T#1S),
					Q => ErrWorkPos);

(* Timeout WorkPos ************************************************)
	tonErrBasePos(	IN := Q_ToBasePos AND (NOT InBasePos OR InWorkPos),
					PT := MAX(PT_Timeout + PT_SensorDamping,PT_Feedback + T#1S),
					Q => ErrBasePos);
					
(*********************************************************************)
	_runtimeChk									:= TRUE;
END_METHOD

METHOD PROTECTED _writeStatus : BOOL
VAR_INPUT
END_VAR


	(* Move *)
	IF Q_ToBasePos AND NOT Q_ToWorkPos AND (NOT InBasePos OR InWorkPos)
	THEN
		Status.0 											:= NOT Options.4;
		Status.1											:= Options.4;
	ELSIF Q_ToWorkPos AND NOT Q_ToBasePos AND (NOT InWorkPos OR InBasePos)
	THEN
		Status.0											:= Options.4;
		Status.1											:= NOT Options.4;
	END_IF              									

	(* BasePos / WorkPos reached*)
	Status.2 												:= SEL(Options.4, InBasePos , InWorkPos);
	Status.3 												:= SEL(Options.4, InWorkPos , InBasePos);
 				        									
	(* Feed ok *)    									
	Status.4 												:= SEL(Options.4, FeedBasePos , FeedWorkPos);
	Status.5 												:= SEL(Options.4, FeedWorkPos , FeedBasePos);
                        									
	(* Ready *)         									
	Status.6												:= NOT Status.7; 
	                    									
	(* Error *)         									
	Status.7 												:= ErrBasePos OR ErrWorkPos OR ErrLogic;
	
	(* Logic error bit **********************************************)
	ErrLogic												:= InBasePos AND InWorkPos AND NOT Options.3;
	
	(* Result *)
	_writeStatus												:= TRUE;
END_METHOD

METHOD PUBLIC enable : BOOL //Return Done = TRUE if WorkPos is TRUE and InWorkPos = TRUE or WorkPos is FALSE and InBasePos is TRUE 
VAR_INPUT
	IN													:	BOOL; //TRUE=WORK / FALSE=BASE
END_VAR
IF IN
THEN
	Enable 													:= THIS^.moveToWorkPos();
ELSE
	Enable 													:= This^.moveToBasePos();
END_IF
END_METHOD

METHOD PUBLIC moveToBasePos : BOOL //Return = Done -> InBasePos
ToWorkPos 									:= Q_ToWorkPos	:= FALSE;
ToBasePos 													:= TRUE;
Q_ToBasePos	 												:= FeedBasePos AND (NOT Options.7 OR NOT InBasePos);
moveToBasePos 									:= Done			:= InBasePos;
Busy														:= NOT Done;
END_METHOD

METHOD PUBLIC moveToWorkPos : BOOL //Return = Done -> InWorkPos
ToBasePos 								:= Q_ToBasePos 		:= FALSE;
ToWorkPos													:= TRUE;
Q_ToWorkPos	 												:= FeedWorkPos AND (NOT Options.7 OR NOT InWorkPos);
moveToWorkPos								:= Done 				:= InWorkPos;
Busy														:= NOT Done;
END_METHOD

METHOD PUBLIC reset : BOOL //Result = reset done
	TonErrWorkPos(IN := FALSE);
	tonErrBasePos(IN := FALSE);
	ErrWorkPos	:= ErrBasePos := ErrLogic						:= FALSE;										
	Status.7 													:= FALSE;
	reset														:= TRUE;
END_METHOD

METHOD PUBLIC switchOff : BOOL
VAR_INPUT
END_VAR
	ToWorkPos	:= FALSE;
	ToBasePos	:= FALSE;
	Done		:= FALSE;
	Busy		:= FALSE;
	Q_ToBasePos	:= FALSE;
	Q_ToWorkPos	:= FALSE;
	switchOff	:= TRUE;
END_METHOD

{attribute 'monitoring' := 'call'}
PROPERTY PUBLIC optDisableLogicError : BOOL
GET
optDisableLogicError := Options.3;
END_GET
SET
Options.3 := optDisableLogicError;
END_SET
END_PROPERTY

{attribute 'monitoring' := 'call'}
PROPERTY PUBLIC optDisableSensorBasepos : BOOL
GET
optDisableSensorBasepos := Options.0;
END_GET
SET
OPtions.0 := optDisableSensorBasepos;
END_SET
END_PROPERTY

{attribute 'monitoring' := 'call'}
PROPERTY PUBLIC optDisableSensorWorkpos : BOOL
GET
optDisableSensorWorkpos := Options.1;
END_GET
SET
OPtions.1 := optDisableSensorWorkpos;
END_SET
END_PROPERTY

{attribute 'monitoring' := 'call'}
PROPERTY PUBLIC optEnableImpulsValveFnc : BOOL
GET
optEnableImpulsValveFnc := Options.7;
END_GET
SET
Options.7 := optEnableImpulsValveFnc;
END_SET
END_PROPERTY

{attribute 'monitoring' := 'call'}
PROPERTY PUBLIC optInvertSensorBasepos : BOOL
GET
optInvertSensorBasepos := Options.5;
END_GET
SET
Options.5 := optInvertSensorBasepos;
END_SET
END_PROPERTY

{attribute 'monitoring' := 'call'}
PROPERTY PUBLIC optInvertSensorWorkpos : BOOL
GET
optInvertSensorBasepos := Options.6;
END_GET
SET
Options.6 := optInvertSensorBasepos;
END_SET
END_PROPERTY

{attribute 'monitoring' := 'call'}
PROPERTY PUBLIC optSwapSensorStatus : BOOL
GET
optSwapSensorStatus := Options.4;
END_GET
SET
OPtions.4 := optSwapSensorStatus;
END_SET
END_PROPERTY

{attribute 'monitoring' := 'call'}
PROPERTY PUBLIC inError : Bool
GET
InError									:= Status.7;
END_GET
END_PROPERTY

{attribute 'monitoring' := 'call'}
PROPERTY public isBusy : bool
GET
isBusy := Busy;
END_GET
END_PROPERTY

{attribute 'monitoring' := 'call'}
PROPERTY isInBasePos : BOOL
GET
isInBasePos := InBasePos;
END_GET
END_PROPERTY

{attribute 'monitoring' := 'call'}
PROPERTY isInWorkPos : BOOL
GET
isInWorkPos := InWorkPos;
END_GET
END_PROPERTY

{attribute 'monitoring' := 'call'}
PROPERTY public isOff : BOOL
GET
isOff := not ToWorkPos and not ToBasePos;
END_GET
END_PROPERTY

{attribute 'monitoring' := 'call'}
PROPERTY PUBLIC noFeed : BOOL
GET
noFeed						:= ToWorkPos and not FeedWorkPos or ToBasePos and not FeedBasePos;
END_GET
END_PROPERTY

{attribute 'monitoring' := 'call'}
PROPERTY Public ok : bool
GET
ok := Done;
END_GET
END_PROPERTY

{attribute 'monitoring' := 'call'}
PROPERTY PUBLIC rCylinder : REFERENCE TO Cylinder
GET
rCylinder REF= This^;
END_GET
END_PROPERTY

{attribute 'monitoring' := 'call'}
PROPERTY simulation : BOOL
GET
simulation := SimulationOn;
END_GET
SET
SimulationOn := simulation;
END_SET
END_PROPERTY

END_FUNCTION_BLOCK

// POUs/IO/Cylinder/I_Cylinder
INTERFACE I_Cylinder EXTENDS I_ActuatorWorkBase

METHOD enable : BOOL //Result value = successful execution of desired action 
VAR_INPUT
	IN							:	BOOL; //TRUE = to Work pos / FLASE = to base pos
END_VAR
END_METHOD

{attribute 'monitoring' := 'call'}
PROPERTY PUBLIC inError : Bool
GET
END_GET
END_PROPERTY

{attribute 'monitoring' := 'call'}
PROPERTY isBusy : BOOL
GET
END_GET
END_PROPERTY

{attribute 'monitoring' := 'call'}
PROPERTY isInBasePos : BOOL
GET
END_GET
END_PROPERTY

{attribute 'monitoring' := 'call'}
PROPERTY isInWorkPos : BOOL
GET
END_GET
END_PROPERTY

METHOD PUBLIC moveToBasePos : BOOL //Return = Done -> InBasePos
END_METHOD

METHOD PUBLIC moveToWorkPos : BOOL //Return = Done -> InWorkPos
END_METHOD

{attribute 'monitoring' := 'call'}
PROPERTY noFeed : BOOL
GET
END_GET
END_PROPERTY

{attribute 'monitoring' := 'call'}
PROPERTY PUBLIC rCylinder : REFERENCE TO Cylinder
GET
END_GET
END_PROPERTY

{attribute 'monitoring' := 'call'}
PROPERTY simulation : BOOL
GET
END_GET
SET
END_SET
END_PROPERTY

METHOD PUBLIC switchOff : BOOL
VAR_INPUT
END_VAR
END_METHOD

END_INTERFACE

// POUs/IO/Cylinder/CylinderExt
{attribute 'no_check'}
//Cylinder with runtime status, extended from FB Cylinder
FUNCTION_BLOCK CylinderExt EXTENDS Cylinder 
VAR_OUTPUT CONSTANT
END_VAR
VAR_INPUT  

END_VAR                                     			
VAR_OUTPUT     			
	RuntimeWP												:	TIME;
	RuntimeBP												:	TIME;
END_VAR
VAR
END_VAR

	(* Cylinder	with runtime status 												*)
	(********************************************************************************)

(* Call super ********************************************************)
	SUPER^();
	
(*********************************************************************)

METHOD PROTECTED _runtimeChk : BOOL
VAR_INPUT
END_VAR
VAR
	memRtBP												:	TIME;
	memRtWP												:	TIME;
END_VAR
(* Record current runtime **********************************************)
	memRtBP													:= tonErrBasePos.ET;
	memRtWP													:= TonErrWorkPos.ET;
	
(* Call time *********************************************************)
	SUPER^._runtimeChk();
	
(* Record last runtime *********************************************)
	IF memRtWP > T#0MS AND NOT tonErrWorkPos.IN AND NOT tonErrWorkPos.Q
	THEN
		RuntimeWP											:= memRtWP;
	END_IF
	
	IF memRtBP > T#0MS AND NOT tonErrBasePos.IN AND NOT tonErrBasePos.Q
	THEN
		RuntimeBP											:= memRtBP;
	END_IF
					
(*********************************************************************)
	_runtimeChk												:= TRUE;

(**********************************************************************)
END_METHOD

END_FUNCTION_BLOCK

// POUs/IO/Cylinder/CylinderType4
{attribute 'no_check'}
//Cylinder with 2x inputs each for work and base position, extended from FB Cylinder
FUNCTION_BLOCK CylinderType4 EXTENDS Cylinder
VAR_OUTPUT CONSTANT
END_VAR
VAR_INPUT  
END_VAR                                     			
VAR_OUTPUT    
{attribute 'displaymode':='binary'}
	ErrInfo													:	BYTE; //.0 BP#1 | .1 BP#2 | .2 WP#1 | .3 WP#2 | .6 Logic Pair#1 | .7 Logic Pair#2 
END_VAR
VAR// IOs 
	SensorBasePos2											: INPUT;
	SensorWorkPos2											: INPUT;
END_VAR

	(* Cylinder	with two inputs for work and base pos each					      	*)
	(* Includes functionblock "INPUT" 												*)
	(********************************************************************************)

(* Write Output *****************************************************)
	IF ToBasePos 	
	THEN
		moveToBasePos();
	ELSIF ToWorkPos AND NOT ToBasePos
	THEN
		moveToWorkPos();
	ELSE
		switchOff();
	END_IF

(* Reedkontakte lesen ***********************************************)
	_readSensors();
	
(* Status *************************************************)
	_writeStatus();
                        	
(* ack Error **********************************************************)
	IF Quit  THEN  reset(); END_IF

(* Timeout  ************************************************)
	_runtimeChk();
	
(*********************************************************************)

METHOD PROTECTED _readSensors : BOOL
VAR_INPUT
END_VAR
(* Call super read sensors first *********************************)
	SUPER^._readSensors();

(* check inputs 2# ************************************************)
	SensorBasePos2(
		Force	:= SensorBasePos.Force ,
		Invert	:= SensorBasePos.Invert,
		PT_ON	:= SensorBasePos.PT_ON,
		PT_OFF	:= SensorBasePos.PT_OFF,
		Q_DIRECT=>,
		Q		=> ,
		Q_RT	=> ,
		Q_FT	=> ,
		IN		=> );


	SensorWorkPos2(
		Force	:= SensorWorkPos.Force,
		Invert	:= SensorWorkPos.Invert,
		PT_ON	:= SensorWorkPos.PT_ON,
		PT_OFF	:= SensorWorkPos.PT_OFF,
		Q_DIRECT=>,
		Q		=> ,
		Q_RT	=> ,
		Q_FT	=> ,
		IN		=> );
		
(* Write status ******************************************)
	InBasePos 									:= SensorBasePos.Q AND SensorBasePos2.Q;
	InWorkPos 									:= SensorWorkPos.Q AND SensorWorkPos2.Q;
	
(* Write error info ***************************************)
	ErrInfo.0									:= TonErrBasePos.Q AND NOT SensorBasePos.Q;
	ErrInfo.1									:= TonErrBasePos.Q AND NOT SensorBasePos2.Q;
	ErrInfo.2									:= TonErrWorkPos.Q AND NOT SensorWorkPos.Q;
	ErrInfo.3									:= TonErrWorkPos.Q AND NOT SensorWorkPos2.Q;

	ErrInfo.6									:= SensorBasePos.Q AND SensorWorkPos.Q;
	ErrInfo.7									:= SensorBasePos2.Q AND SensorWorkPos2.Q;
	
(**************************************************************)
	_readSensors								:= TRUE;
	
(*****************************************************************)
END_METHOD

END_FUNCTION_BLOCK

// POUs/IO/Drives/CoE/EL72xx/AxDriveCoE_EL72xxParam
{attribute 'no_check'}
//FB template to read and write parameter
//The FB can be enherided and derivatived methods of SeqRead/SeqWrite used for application specific parameter.
//The extended methods need to call the super class at the beginning and return true if execution will be finished. The allowed states for new parameter are 1..99
FUNCTION_BLOCK AxDriveCoE_EL72xxParam EXTENDS AxRWParaBase
VAR_OUTPUT CONSTANT
END_VAR                                 					
VAR_INPUT                               					
	AdsAddr													: 	AMSADDR; //Terminal AMS Net Addr.     
	Channel													:	USINT := 0; //Drive channel 0 or 1                                    	                                        	
	SetKvPosition											:	LREAL; //(rad/s)rad - e.g. 10.0		0x8010:17
	SetKpVelocity											:	LREAL; //mA/(rad/s) - e.g. 0.058	0x8010:15
	SetTnVelocity											:	LREAL; //0.1ms 		- e.g. 0.015	0x8010:14
END_VAR 
VAR_IN_OUT
END_VAR                               					
VAR_OUTPUT
	DeviceType												:	STRING(15); //0x1008:0 -e.g. EL7211-9014
	MotorSN													:	STRING(15); //0x9009:13 - if available
	KvPosition												:	LREAL;
	KpVelocity												:	LREAL;
	TnVelocity												:	LREAL;	
END_VAR                         	
VAR
(* Cache ************************************************************)

(* Trigger **********************************************************)

(* Timer ******************************************************************)

(* FBs ***************************************************************)
	CoEWrite												: FB_EcCoESdoWriteEx := (tTimeout := DEFAULT_ADS_TIMEOUT); //CoE read
	CoERead													: FB_EcCoeSdoReadEx := (tTimeout := DEFAULT_ADS_TIMEOUT);

(* Dummy memory **********************************************************)
END_VAR

	(* Read/Write drive parameter														*)
	(************************************************************************************)

(* Execute ***************************************************************************************)
	SUPER^();

(*************************************************************************************************)

PROPERTY PROTECTED deviceAddrIsValid : BOOL
GET
deviceAddrIsValid := AdsAddr.port > 0;
END_GET
END_PROPERTY

METHOD PROTECTED getValue : BOOL //Return value = TRUE if execution finished and state incremented 
VAR_INPUT
	Index						:	WORD;
	SubIndex					:	BYTE;
	Len							:	UDINT;
	pActValue					:	PVOID; //Address of variable for actual value
	pSetValue					:	PVOID; //Address of variable for ser value variable, can be zero if no corresponding SetVariable exists
	CompleteAccess				:	BOOL;
END_VAR
CoERead(bExecute := TRUE , nIndex := Index ,nSubIndex := SubIndex ,pDstBuf := pActValue ,cbBufLen := Len, bCompleteAccess  := CompleteAccess);
IF NOT CoERead.bBUSY 	
THEN
	IF NOT CoERead.bError
	THEN
		IF pSetValue <> 0 THEN MEMCPY(pSetValue, pActValue, Len); END_IF
		state 												:= state + 1; 
	ELSE
		Busy												:= FALSE;
		Error												:= TRUE;
		ErrorId												:= CoERead.nErrId;
		ErrorText											:= CONCAT('Error read parameter in state:' , TO_STRING(state * -1));
		ErrorText											:= CONCAT(ErrorText , ' Id:');
		ErrorText											:= CONCAT(ErrorText , TO_STRING(ErrorId));
		State												:= 9999;
	END_IF
	CoERead(bExecute := FALSE);
	getValue												:= TRUE;
END_IF
END_METHOD

METHOD PROTECTED seqRead : BOOL //Return value = TRUE if execution finished 
VAR_IN_OUT
	state							:	INT;
END_VAR

(* Sequence read parameter **********************************)
	CASE state OF
	1..99: //Read application specific parameter  
		SeqRead												:= TRUE;
		
	1001: (* Init step ******************************************************)
		CoERead(bExecute := FALSE, sNetId:= F_CreateAmsNetId(nIds := AdsAddr.netId), nSlaveAddr:= AdsAddr.port);
		IF NOT CoERead.bBusy
		THEN
			state											:= state + 1;	
		END_IF
		
	1002: (* Device name *************************************************************************************)
		IF LEN(DeviceType) > 0 AND NOT CoERead.bBusy
		THEN
			state											:= state + 1;
		ELSE
			getValue(Index:= 16#1008,	Subindex := 16#0,	LEN := SIZEOF(DeviceType),	pActValue := ADR(DeviceType),	pSetValue := 0, completeAccess := FALSE);
		END_IF

	1003: (* Motor SN *************************************************************************************)		
		IF LEN(MotorSN) > 0 AND NOT CoERead.bBusy
		THEN
			state											:= state + 1;
		ELSE
			getValue(Index:= 16#9009,	Subindex := 16#03,	LEN := SIZEOF(MotorSN),		pActValue := ADR(MotorSN),	pSetValue := 0, completeAccess := FALSE);
		END_IF
			
	1004: (* kv position *******************************************)
		IF getValue(Index:= 16#8010,	Subindex := 16#17,	LEN := SIZEOF(_UDINT),		pActValue := ADR(_UDINT),	pSetValue := 0, completeAccess := FALSE)
		THEN
			KvPosition := SetKvPosition						:= SEL(Error, TO_LREAL(_UDINT) * 1.0, 0.0); 
		END_IF
	
	1005: (* Kp velocity *******************************************)
		IF getValue(Index:= 16#8010,	Subindex := 16#15,	LEN := SIZEOF(_UDINT),		pActValue := ADR(_UDINT),	pSetValue := 0, completeAccess := FALSE)
		THEN
			KpVelocity := SetKpVelocity						:= SEL(Error, TO_LREAL(_UDINT) * 0.001, 0.0);
		END_IF
		
	1006: (* Tn velocity ********************************************)
		IF getValue(Index:= 16#8010,	Subindex := 16#14,	LEN := SIZEOF(_UDINT),		pActValue := ADR(_UDINT),	pSetValue := 0, completeAccess := FALSE)
		THEN
			TnVelocity := SetTnVelocity						:= SEL(Error, TO_LREAL(_UDINT) * 0.0001, 0.0);
		END_IF
	ELSE
		state												:= 1;
	END_CASE

(***********************************************************************************)
END_METHOD

METHOD PROTECTED seqWrite : BOOL //Return value = TRUE if execution finished 
VAR_IN_OUT
	state							:	INT;
END_VAR
(* Sequence write parameter *********************************************)
	CASE state OF
	1..99: //Write application specific parameter  
		SeqWrite											:= TRUE;
		
	1001: (* Init step ******************************************************)
		CoEWrite(bExecute := FALSE, sNetId:= F_CreateAmsNetId(nIds := AdsAddr.netId), nSlaveAddr:= AdsAddr.port);
		IF NOT CoEWrite.bBusy
		THEN
			state											:= state + 1;	
		END_IF
	
	1002: (* Kv position *************************************************************************************)
		_UDINT												:= TO_UDINT(SetKvPosition * 1.0);
		IF setValue(Index:= 16#8010,	Subindex := 16#17,	LEN := SIZEOF(_UDINT),		pActValue := 0,		pSetValue := ADR(_UDINT) , completeAccess := FALSE)
		THEN
			KvPosition										:= SetKvPosition;
		END_IF
		
	1003: (* Kp velocity ****************************************)
		_UDINT											:= TO_UDINT(SetKpVelocity * 1000.0);
		IF setValue(Index:= 16#8010,	Subindex := 16#15,	LEN := SIZEOF(_UDINT),		pActValue := 0,		pSetValue := ADR(_UDINT), completeAccess := FALSE)
		THEN
			KpVelocity										:= SetKpVelocity;
		END_IF

	1004: (* Tn velocity **********************************)
		_UDINT											:= TO_UDINT(SetTnVelocity * 10000.0);
		IF setValue(Index:= 16#8010,	Subindex := 16#14,	LEN := SIZEOF(_UDINT),		pActValue := 0,		pSetValue := ADR(_UDINT), completeAccess := FALSE)
		THEN
			TnVelocity										:= SetTnVelocity;
		END_IF	
	ELSE
		state												:= 1;
	END_CASE

(************************************************************************************)
END_METHOD

METHOD PROTECTED setValue : BOOL //Return value = TRUE if execution finished and state incremented 
VAR_INPUT
	Index						:	Word;
	SubIndex					:	BYTE;
	Len							:	UDINT;
	pActValue					:	PVOID; //Address of variable for actual value, can be zero if no corresponding acual value variable exists
	pSetValue					:	PVOID; //Address of variable for set value variable
	CompleteAccess				:	BOOL;
END_VAR


IF pActValue <> 0 AND pSetValue <> 0 AND_THEN MEMCMP(pSetValue, pActValue, Len) = 0
THEN //Skip write parameter if set and actual value are equel
	state													:= state + 1;	
	setValue												:= TRUE;
ELSE
	CoEWrite(bExecute := TRUE, nIndex := Index ,nSubIndex := SubIndex , pSrcBuf := pSetValue ,cbBufLen := Len , bCompleteAccess := CompleteAccess );
	IF NOT CoEWrite.bBusy
	THEN
		IF NOT CoEWrite.bError
		THEN
			IF pActValue <> 0 THEN MEMCPY(pActValue, pSetValue, Len); END_IF	
			state											:= state + 1;
		ELSE
			Busy											:= FALSE;
			Error											:= TRUE;
			ErrorId											:= CoEWrite.nErrId;
			ErrorText										:= CONCAT('Error write parameter in state:' , TO_STRING(state * -1));
			ErrorText										:= CONCAT(ErrorText , ' Id:');
			ErrorText										:= CONCAT(ErrorText , TO_STRING(ErrorId));
			State											:= 9999;
		END_IF
		CoEWrite(bExecute := FALSE);
		setValue											:= TRUE;
	END_IF		
END_IF
END_METHOD

END_FUNCTION_BLOCK

// POUs/Motion/TF50xx-NC/00_Base/AxRWParaBase
{attribute 'no_check'}
//FB template to read and write parameter
//The FB can be enherided and derivatived methods of SeqRead/SeqWrite used for application specific parameter.
//The extended methods need to call the super class at the beginning and return true if execution will be finished. The allowed states for new parameter are 1..99
FUNCTION_BLOCK AxRWParaBase EXTENDS FbBase
VAR_OUTPUT CONSTANT
	FNC_READ												:	INT := 0;
	FNC_WRITE												:	INT := 1;
END_VAR                                 					
VAR_INPUT                               					
	Fnc														:	INT (FNC_READ..FNC_WRITE) := FNC_READ;    
	EnableAutoInit											:	BOOL := TRUE; (* FB will start internal init (read all parameter) at first call if set to true   *)                                	                                        	
END_VAR                                 					
VAR_OUTPUT                              										
	InitDone												:	BOOL := FALSE; (* Parameter initalisation done - Set parameter are initaliced by active values *)
	ErrorText												:	STRING := '';
END_VAR                         	


VAR
(* Zwischenspeicher ************************************************************)
	MemFnc													:	INT := -1;
	LastError												:	STRING;
	
(* Deklaration Trigger **********************************************************)

(* Zeiten ******************************************************************)

(* Bausteine ***************************************************************)

(* Dummy Speicher **********************************************************)
	_INT													: INT;
	_UINT													: UINT;
	_UDINT													: UDINT;
	_LREAL													: LREAL;
	_DWORD													: DWORD;
END_VAR

	(************************************************************************************)
	(*																					*)
	(*		B E C K H O F F   N E W   A U T O M A T I O N   T E C H N O L O G Y    		*)
	(*																					*)
	(*		Eiserstr.5	D-33415 Verl	Germany	phone:	+49-5246-0	www.Beckhoff.Com	*)
    (*																					*)
    (*		Bausteinbeschreibung	:	Read/Write parameter template					*)
	(*																					*)
	(************************************************************************************)

(* Execute ***************************************************************************************)
	rtExecute(CLK := Execute);
	IF(rtExecute.Q OR NOT InitDone AND EnableAutoInit)
		AND MemFnc < 0
	THEN
		MemFnc 												:= SEL(Fnc = FNC_WRITE AND InitDone, FNC_READ , FNC_WRITE) ;
		Busy												:= TRUE;
		Done												:= FALSE;
		Error												:= FALSE;
		ErrorID												:= 0;
		LastError											:= ErrorText;
		ErrorText											:= '';
	END_IF

(* Call Method ***********************************************************************************)
	CASE MemFnc OF
	FNC_READ:
		Read(Execute);

	FNC_WRITE:
		Write(Execute);

	-1:
		IF NOT Execute
		THEN
			Busy											:= FALSE;
			Done											:= FALSE;
			Error											:= FALSE;
			ErrorID											:= 0;
			LastError										:= ErrorText;
			ErrorText										:= '';
		END_IF                              				
	ELSE                                    				
		Busy												:= FALSE;
		Done												:= FALSE;
		Error												:= Execute;
		ErrorID												:= E_AdsErr.DEVICE_INVALIDPARM;
		ErrorText											:= CONCAT('Prg error, invalid MemFnc value ', TO_STRING(MemFnc));
	END_CASE                                    			
	
(*************************************************************************************************)

PROPERTY PROTECTED deviceAddrIsValid : BOOL
GET
deviceAddrIsValid := TRUE;
END_GET
END_PROPERTY

METHOD PUBLIC FINAL read : BOOL //Return value = TRUE if busy
VAR_INPUT
	Execute													: BOOL;
END_VAR
IF MemFnc = FNC_WRITE AND busy
THEN
	Busy													:= FALSE;
	Error													:= TRUE;
	ErrorId													:= E_AdsErr.DEVICE_BUSY;
	ErrorText												:= CONCAT('Error read parameter in state:' , TO_STRING(state * -1));
	ErrorText												:= CONCAT(ErrorText , ' write parameter is active, Id:');
	ErrorText												:= CONCAT(ErrorText , TO_STRING(ErrorId));
	MemFnc													:=  -1;
	Read													:= FALSE;
ELSE
	MemFnc													:= FNC_READ;
	THIS^.Execute											:= Execute;

	(* Parameter lesen Statemaschine *************************************************************************)
	CASE state OF
	0:	(* Init *)	
		IF(Execute OR NOT InitDone AND EnableAutoInit AND deviceAddrIsValid)
		THEN
		
			IF deviceAddrIsValid
			THEN
				Busy										:= TRUE;
				Done										:= FALSE;
				Error										:= FALSE;
				ErrorId 									:= 0;
				ErrorText									:= '';
				state										:= 1001;
			ELSE
				Busy										:= FALSE;
				Done										:= FALSE;
				Error										:= TRUE;
				ErrorId 									:= 24; //Invalid ads port 
				ErrorText									:= CONCAT('Error read parameter in state:' , TO_STRING(state * -1));
				ErrorText									:= CONCAT(ErrorText , '| ID/Addr. of device invalid');
				state										:= 9999;			
			END_IF
		ELSE                        						
			Busy											:= FALSE;
			Done											:= FALSE;
			Error											:= FALSE;
			ErrorId 										:= 0;
			ErrorText										:= '';
		END_IF

	1..99,1001..1099: (* Call sequence read *)
		IF SeqRead(state)
		THEN
			state											:= 9999;	
			InitDone										:= TRUE;
			Done											:= NOT Error;
			Busy											:= FALSE;		
		END_IF
             				
	9999: (* Last state execution finished *****************************)
		IF NOT Execute 
		THEN
			Busy											:= FALSE;
			Done											:= FALSE;
			Error											:= FALSE;
			ErrorId 										:= 0;
			ErrorText										:= '';
		END_IF
		
	ELSE (* Case else *)	
		Busy												:= FALSE;
		Error												:= TRUE;
		ErrorId												:= E_AdsErr.DEVICE_INVALIDSTATE;
		ErrorText											:= CONCAT('Error read parameter; invalid state:' , TO_STRING(state));
		ErrorText											:= CONCAT(ErrorText , ' Id:');
		ErrorText											:= CONCAT(ErrorText , TO_STRING(ErrorId));
		State												:= 9999;
	END_CASE

	(* Reset state to zero if Execute is set back to false *)
	IF NOT Execute AND NOT busy
	THEN
		MemFnc												:=  -1;
		state 												:= 0;
	END_IF
	
	Read													:= Busy; //Return;
END_IF	

(****************************************************************************************************************)
END_METHOD

METHOD PROTECTED seqRead : BOOL //Return value = TRUE if execution finished 
VAR_IN_OUT
	state							:	INT;
END_VAR
CASE state OF
1,1001:
(* Example
		IF getValue(IDxGrp:= 16#5100,	IDxOffs := 16#9,	LEN := SIZEOF(uiValue),	pActValue := ADR(uiValue),  pSetValue := 0)
		THEN
			SetRefFlag :=RefFlag							:= TO_BOOL(uiValue);
		END_IF
*)
	SeqRead													:= TRUE;
ELSE
	SeqRead													:= TRUE;
END_CASE
END_METHOD

METHOD PROTECTED seqWrite : BOOL //Return value = TRUE if execution finished 
VAR_IN_OUT
	state							:	INT;
END_VAR
CASE state OF
1,1001:
(* Example 
	setValue(IDxGrp:= 16#4000,	IDxOffs := 16#102,	LEN := SIZEOF(SetDec), pActValue := ADR(Dec),	pSetValue := ADR(SetDec));
*)
	SeqWrite												:= TRUE;
ELSE
	SeqWrite												:= TRUE;
END_CASE
END_METHOD

METHOD PUBLIC FINAL write : BOOL //Return value = TRUE if busy
VAR_INPUT
	Execute													:	BOOL;
END_VAR
IF MemFnc = FNC_READ AND busy
THEN
	Busy													:= FALSE;
	Error													:= TRUE;
	ErrorId													:= E_AdsErr.DEVICE_BUSY;
	ErrorText												:= CONCAT('Error write parameter in state:' , TO_STRING(state * -1));
	ErrorText												:= CONCAT(ErrorText , ' read parameter is active, Id:');
	ErrorText												:= CONCAT(ErrorText , TO_STRING(ErrorId));
	MemFnc													:=  -1;
	Write													:= FALSE;
ELSE
	MemFnc													:= FNC_WRITE;
	THIS^.Execute											:= Execute;

(* Parameter schreiben ************************************************************************************************)
	(* Parameter schreiben Statemaschine *)
	CASE state OF
	0:	(* Init *)	
		IF Execute 
		THEN
			IF deviceAddrIsValid
			THEN
				Busy										:= TRUE;
				Done										:= FALSE;
				Error										:= FALSE;
				ErrorId 									:= 0;
				state										:= 1001;
			ELSE
				Busy										:= FALSE;
				Done										:= FALSE;
				Error										:= TRUE;
				ErrorId 									:= 24; //Invalid ads port 	
				ErrorText									:= CONCAT('Error write parameter in state:' , TO_STRING(state * -1));
				ErrorText									:= CONCAT(ErrorText , '| ID/Addr. of device invalid');
				state										:= 9999;			
			END_IF                  						
		ELSE 
			Busy											:= FALSE;
			Done											:= FALSE;
			Error											:= FALSE;
			ErrorId 										:= 0;
			ErrorText										:= '';
		END_IF
		
	1..99,1001..1099: (* Call sequence write *)
		IF SeqWrite(state)
		THEN
			Done											:= NOT Error;
			Busy											:= FALSE;
			state											:= 9999;			
		END_IF	
		
	9999: (* Last state execution finished *****************************)
		IF NOT Execute 
		THEN
			Busy											:= FALSE;
			Done											:= FALSE;
			Error											:= FALSE;
			ErrorId 										:= 0;
			ErrorText										:= '';
		END_IF
		
	ELSE (* Case else *)	
		Busy												:= FALSE;
		Error												:= TRUE;
		ErrorId												:= E_AdsErr.DEVICE_INVALIDSTATE;
		ErrorText											:= CONCAT('Error write parameter; invalid state:' , TO_STRING(state));
		ErrorText											:= CONCAT(ErrorText , ' Id:');
		ErrorText											:= CONCAT(ErrorText , TO_STRING(ErrorId));
		State												:= 9999;
	END_CASE

	(* Reset state to zero if Execute is set back to false *)
	IF NOT Execute AND NOT busy
	THEN
		MemFnc												:=  -1;
		state 												:= 0;
	END_IF
	
	Write													:= Busy; //Return;
END_IF
END_METHOD

END_FUNCTION_BLOCK

// POUs/IO/Drives/CoE/EL72xx/CiA_DS402StatuswordEx7xxx
FUNCTION_BLOCK CiA_DS402StatuswordEx7xxx EXTENDS CiA_DS402Statusword
VAR_INPUT
END_VAR
VAR_OUTPUT	

	TxPDOToggle				: BOOL; // Bit 10: Following error occured
	FollowCmdValue			: bool;  //Bit 12: Drive follows command (CSP/CSV)
	InputCycleCounter		: BOOL; // Bit 13: 
END_VAR

METHOD PUBLIC readStatusword : BOOL
VAR_INPUT
	Statusword 		:	UINT;
END_VAR
SUPER^.readStatusword(Statusword);

TxPDOToggle													:= Statusword.10;
FollowCmdValue												:= Statusword.12;
InputCycleCounter											:= Statusword.13 ;
	
readStatusword												:= TRUE;
END_METHOD

END_FUNCTION_BLOCK

// POUs/IO/Drives/CoE/CiA_DS402Statusword
FUNCTION_BLOCK CiA_DS402Statusword
VAR_INPUT
END_VAR
VAR_OUTPUT	
	ReadyToSwitchOn			: BOOL; //Bit 0: Ready TO switch on	- - Controlled by state machine
	SwitchedOn				: BOOL; //Bit 1: Switched on - Controlled by state machine
	OperationEnabled		: BOOL; //Bit 2: Operation enabled - Controlled by state machine
	Fault					: BOOL; //Bit 3: Drive fault active
	VoltageEnabled			: BOOL; //Bit 4 - Manufacturer specific / Voltage enabled
	QuickStopInverse		: BOOL; // Bit 5: False = Quick stop active (inverse signal)- Controlled by state machine
	SwitchOnDisabled		: BOOL; // Bit 6: Switch in disabled - Controlled by state machine
	Warning					: BOOL; // Bit 7: Warning active
//Manufacturer specific_Bit8
	RemoteActive			: BOOL;  // Bit 9: ManufacturerSpecific_Bit9, commonly used for control over network (EtherCAT) active
//	TargetReached			: BOOL; // Bit 10 commonly used for in target position, velocity in pp or pv mode
//	TxPDOToggle				: BOOL; // Bit 10: TxPDOToggle (An-/Abwahl über 0x8010:01)
	InternalLimitActive		: BOOL; // Bit 11: Internal limit active
//Operation mode specific_Bit12	- pp = Set-point acknowledge, pv = standstill, hm = Homing attained, csp = following set pos., csv following set velo
//Operation mode specific_Bit13 - pp = Following error, pv = N/A, hm = Homing error, csp = Following error, csv = N/A
//Manufacturer specific_Bit14
//Manufacturer specific_Bit15

	State					: eCiA_DS402_STATUS_STATE; // Device state
END_VAR

METHOD PUBLIC readStatusword : BOOL
VAR_INPUT
	Statusword 					:	UINT;
END_VAR
//Status bits
ReadyToSwitchOn												:= Statusword.0 ;
SwitchedOn													:= Statusword.1 ;
OperationEnabled											:= Statusword.2 ;
Fault														:= Statusword.3 ;
VoltageEnabled												:= Statusword.4 ;
QuickStopInverse											:= Statusword.5 ;
SwitchOnDisabled											:= Statusword.6 ;
Warning														:= Statusword.7 ;

RemoteActive												:= Statusword.9 ;

InternalLimitActive											:= Statusword.11;


//State
IF NOT ReadyToSwitchOn 
THEN
	IF SwitchOnDisabled
	THEN
		state												:= eCiA_DS402_STATUS_STATE.SWITCH_ON_DISABLED;
	ELSE
		state												:= eCiA_DS402_STATUS_STATE.NOT_READY_TO_SWITCH_ON;
	END_IF
ELSIF Fault
THEN
	IF ReadyToSwitchOn AND SwitchedOn AND OperationEnabled
	THEN
		state												:= eCiA_DS402_STATUS_STATE.FAULT_REACTION_ACTIVE;
	ELSE
		state												:= eCiA_DS402_STATUS_STATE.FAULT_ACTIVE;
	END_IF
ELSE 
	IF QuickStopInverse
	THEN
		state												:= eCiA_DS402_STATUS_STATE.READY_TO_SWITCH_ON;
		IF SwitchedOn
		THEN
			state											:= eCiA_DS402_STATUS_STATE.SWITCHED_ON;
			IF OperationEnabled
			THEN
				state										:= eCiA_DS402_STATUS_STATE.OPERATION_ENABLED;
			END_IF
		END_IF
	ELSE //Quick stop active
		IF SwitchedOn AND OperationEnabled
		THEN
			state											:= eCiA_DS402_STATUS_STATE.QUICK_STOP_ACTIVE;
		ELSIF SwitchOnDisabled
		THEN
			state											:= eCiA_DS402_STATUS_STATE.SWITCH_ON_DISABLED;
		ELSE
			state 											:= eCiA_DS402_STATUS_STATE.NOT_READY_TO_SWITCH_ON;
		END_IF
	END_IF
END_IF

readStatusword												:= TRUE;
END_METHOD

END_FUNCTION_BLOCK

// POUs/IO/Drives/CoE/AxDriveCoE
{attribute 'no_check'}
//CoE Drive status and diagnosis
//Attention: "SwitchedOn" will be only true if bit 12 "FollowCmdValue" of statusword is used by drive
FUNCTION_BLOCK AxDriveCoE EXTENDS AxDriveBase     
VAR CONSTANT								
END_VAR                  						
VAR_INPUT                           						
	BrakeUnlock												:	BOOL := FALSE;
END_VAR
VAR_IN_OUT
END_VAR
VAR_OUTPUT
	BrakeUnlocked											:	BOOL;
	Status													:	CiA_DS402Statusword;	
	InfoData1										AT %I*	:	UINT;
	InfoData2										AT %I*	:	UINT;
END_VAR                             						
VAR
END_VAR
VAR
(* Cache *********************************************************************)

	// CoE Diagmessage
	StatusTrig												: BYTE;
	MemStatusTrig											: BYTE;
	
(* Timer ********************************************************************************)
  	readDiagDelay											: TON := (PT := T#50MS);
                                  						
(* Trigger ******************************************************************************)


(* Function blocks ****************************************************************************)
	ReadCoEDiagMsg											: EcCoEReadNewestDiagMsg := (Timeout := DEFAULT_ADS_TIMEOUT);	
	CoEWrite												: FB_EcCoeSdoWriteEx := (tTimeout := DEFAULT_ADS_TIMEOUT);	

(* Dummy Speicher **********************************************************)
END_VAR

	(* CoE Drive																		*)
	(************************************************************************************)

(* abort function-call if the reference is invalid *****************************)
IF NOT __ISVALIDREF(rAxis) 
THEN
	Fault													:= TRUE;
	SwitchedOn												:= FALSE;
	Ready													:= FALSE;
	RETURN;         										
END_IF

(* Call super class ****************************************************)
	SUPER^(); 
	
(* Read Statusword ********************************************************)	
	IF rAxis.Status.OpMode.SimulationAxis
	THEN
		IF rAxis.PlcToNc.ControlDWord.0
		THEN
			Status.readStatusword(TO_UINT(eCiA_DS402_STATUS_STATE.OPERATION_ENABLED));
		ELSE
			Status.readStatusword(TO_UINT(eCiA_DS402_STATUS_STATE.SWITCHED_ON));	
		END_IF
	ELSE
		Status.readStatusword(Statusword);
	END_IF			
	
	(* EL72xx DS402 Statusword
		Bit 0 : Ready to switch on
		Bit 1 : Switched on
		Bit 2 : Operation enabled
		Bit 3 : Fault
		Bit 4 : reserved
		Bit 5 : Quick stop (inverse)
		Bit 6 : Switch on disabled
		Bit 7 : Warning
		Bit 8 + 9 : reserved
		Bit 10 : TxPDOToggle (An-/Abwahl über 0x60DA)
		Bit 11 : Internal limit active
		Bit 12 : (drive follows command value)
		Bit 13 - 15 : reserved *)
		
(* DriveStatusBits ***********************************************)
	Fault													:= Status.Fault
																OR rAxis.NcToPlc.StateDWord.28 (* DriveDeviceError *)
																OR rAxis.NcToPlc.StateDWord.30; (* IODataInvalid *)
            												
	Ready 													:= NOT Fault
																AND(Status.ReadyToSwitchOn OR Status.SwitchedOn);

	SwitchedOn												:= Status.SwitchedOn AND NOT Fault;

	
(* manual override brake ********************************************************)
	IF (BrakeUnlock XOR BrakeUnlocked)
		OR CoEWrite.bBusy
	THEN
		BrakeUnlocked										:= BrakeUnlock;
		CoEWrite(
			bExecute	:= NOT CoEWrite.bBusy AND NOT rAxis.NcToPlc.StateDWord.30 AND AdsAddr.port > 0 AND NOT rAxis.Status.OpMode.SimulationAxis,
			sNetId		:= F_CreateAmsNetId(nIds :=AdsAddr.netId),
			nSlaveAddr	:= AdsAddr.port, 
			nIndex		:= 16#8012, 
			nSubIndex	:= 16#1, 
			pSrcBuf		:= ADR(BrakeUnlocked), 
			cbBufLen	:= SIZEOF(BrakeUnlocked));
	END_IF
	
(* Read diagnoses ***********************************************************)
	StatusTrig.0											:= NOT Status.ReadyToSwitchOn;
	StatusTrig.1											:= Status.Fault;
	StatusTrig.2											:= Status.Warning AND NOT Status.Fault;
	
	CASE state OF
	0: // Read subindex of the newest diagnosis message
		
		readDiagDelay(IN := StatusTrig <> MemStatusTrig AND NOT rAxis.Status.OpMode.SimulationAxis AND AdsAddr.port > 0);
	
		IF readDiagDelay.Q
		THEN
			ReadCoEDiagMsg( Execute:= FALSE,  AdsAddr:= AdsAddr);
				
			IF NOT ReadCoEDiagMsg.Busy
			THEN
				MemStatusTrig 								:= StatusTrig; 
				readDiagDelay(IN := FALSE);			
				state 										:= state + 1;
			END_IF
		END_IF
	1: // read newest message
		ReadCoEDiagMsg( Execute:= TRUE,  AdsAddr:= AdsAddr);
		IF NOT ReadCoEDiagMsg.Busy
		THEN
			IF ReadCoEDiagMsg.Error
			THEN
				state										:= 0;
			ELSE	
				state										:= 0;			
			END_IF
			ReadCoEDiagMsg(Execute := FALSE);		
		END_IF
		
	END_CASE
	
(******************************************************************************)

END_FUNCTION_BLOCK

// POUs/IO/Drives/AxDriveBase
{attribute 'no_check'}
FUNCTION_BLOCK AxDriveBase EXTENDS EcSlaveInfoDataExt IMPLEMENTS I_AxDriveBase
VAR CONSTANT         	
END_VAR  
VAR_INPUT
	rAxis													:	REFERENCE TO AXIS_REF := 0; //Reference to NC-Axis REF
END_VAR                     					
VAR_IN_OUT                  					
END_VAR                     					
VAR_OUTPUT                  					
	Fault													:	BOOL; (* Drive Error *)
	SwitchedOn												:	BOOL; (* Drive enabled *)
	Ready													:	BOOL; (* Drive Ready *)
{attribute 'displaymode':='binary'}    
	Statusword										AT %I* 	:	UINT; //Link to the drive status word after linking the NC
	Channel											AT %I*	:	USINT;
END_VAR                     					                   					
VAR                         				

END_VAR
VAR

(* Cache *********************************************************************)
	State													:	INT; //State machine 

(* Timer ********************************************************************************)

(* Trigger ******************************************************************************)

(* Instance ****************************************************************************)
	
(* Dummy Speicher **********************************************************)
END_VAR

	(* Drive base information															*)
	(************************************************************************************)
	
	SUPER^();

PROPERTY PUBLIC rAxDrive : REFERENCE TO AxDriveBase
GET
rAxDrive REF= This^;
END_GET
END_PROPERTY

PROPERTY Public rInfoData : reference to EcSlaveInfoData
GET
rInfoData REF= THis^;
END_GET
END_PROPERTY

END_FUNCTION_BLOCK

// POUs/IO/Drives/I_AxDriveBase
INTERFACE I_AxDriveBase EXTENDS __SYSTEM.IQueryInterface

PROPERTY PUBLIC rAxDrive : REFERENCE TO AxDriveBase
GET
END_GET
END_PROPERTY

END_INTERFACE

// POUs/IO/Drives/CoE/AxDriveCoE_wEvents
{attribute 'no_check'}
//Drive 
FUNCTION_BLOCK AxDriveCoE_wEvents EXTENDS AxDriveCoE   
VAR_OUTPUT CONSTANT
{attribute 'displaymode':='binary'}  
	OPTION_DISABLE_INT_LIMIT_WARNING						:	BYTE := 2#0000_0001;
{attribute 'displaymode':='binary'}  
	OPTION_DISABLE_REMOTE_CNTR_NOT_ACTIVE					:	BYTE := 2#0000_0010;	
END_VAR                  						
VAR_INPUT                           						
	EnableEvent												:	BOOL := TRUE;
	{attribute 'displaymode':='binary'}  
	Options													:	BYTE := 0;
	ConfirmTrig												:	BOOL := FALSE; (* Reset event *)
	SourceId												:	UDINT := 102200; //CoE Drive default multisource Id + Ax id
	Name													:	STRING(30) := '';
	ErrorLimitPos											:	BOOL := FALSE;
	ErrorLimitNeg											:	BOOL := FALSE;
END_VAR
VAR_IN_OUT
END_VAR
VAR_OUTPUT
	EventStatus												:	DWORD;
	NoOfActiveEvents										:	INT;
END_VAR                             						
VAR

END_VAR
VAR
(* Cache *********************************************************************)
	
(* Timer ********************************************************************************)
                                						
(* Trigger ******************************************************************************)


(* Function blocks ****************************************************************************)
	
	Event													: EventHandlingGrp10;
	EventDiagMessage										: EventHandling;

(* Dummy Speicher **********************************************************)
	i														: INT := 0 ;

END_VAR

	(* CoE Drive with diag and eventlogger implementation								*)
	(************************************************************************************)

(* call super ***********************************************************************)
	SUPER^();

(* trigger events ************************************************)
	_callEvents();

(*****************************************************************)

METHOD _callEvents : BOOL
VAR_INPUT
END_VAR
(* Check if msg activ and init some parameter ***********************)
	IF Event.no[1].Text2 <> Name AND Name <> '' OR Event.no[1].Text2 = '' AND rAxis.NcToPlc.AxisId <> 0
	THEN
		Event.no[1].eClass 									:= TC2_SYSTEM.TCEVENTCLASS_STATEINFO;
		Event.no[3].eClass 									:= TC2_SYSTEM.TCEVENTCLASS_WARNING;
		Event.no[4].eClass 									:= TC2_SYSTEM.TCEVENTCLASS_WARNING;
		Event.no[5].eClass 									:= TC2_SYSTEM.TCEVENTCLASS_STATEINFO;
		Event.no[6].eClass 									:= TC2_SYSTEM.TCEVENTCLASS_STATEINFO;
		Event.no[7].eClass 									:= TC2_SYSTEM.TCEVENTCLASS_STATEINFO;
		
		(* Init axisname *)
		FOR i := Event.MIN_EVENT TO Event.MAX_EVENT DO
		(*	Event.no[i].Text1								:= '';*)
			Event.no[i].Text2								:= SEL(LEN(name)>1,CONCAT('Axis id:',DWORD_TO_STRING(rAxis.NcToPlc.AxisId)),name);			
		END_FOR
		EventDiagMessage.Text2								:= Event.no[1].Text2;
	END_IF

(* workl Event Ctrl *************************************************)
	Event(
		ConfirmTrig 	:= ConfirmTrig,
		Disable			:= rAxis.NcToPlc.AxisId = 0 OR NOT EnableEvent,
		SourceId		:= SourceId + rAxis.NcToPlc.AxisId);
		

(* Event diag message ***************************************************)
	CASE ReadCoEDiagMsg.MsgSeverity OF
	0: // Info message
		EventDiagMessage.eClass 								:= TCEVENTCLASS_MESSAGE;
	1: // warning
		EventDiagMessage.eClass 								:= TCEVENTCLASS_WARNING;
	2: // error message
		EventDiagMessage.eClass 								:= TCEVENTCLASS_ALARM;
	ELSE // unknown type
		EventDiagMessage.eClass 								:= TCEVENTCLASS_NONE;
	END_CASE
				
	EventDiagMessage(
		Flag			:= state = 0 AND ReadCoEDiagMsg.TextId <> 0 AND (Status.Fault OR Status.Warning) AND NOT Event.Disable,
		ConfirmTrig 	:= ConfirmTrig OR NOT EventDiagMessage.Flag AND EventDiagMessage.State <> TCEVENTSTATE_INVALID,
		MsgId			:= ReadCoEDiagMsg.TextId,
		SourceId		:= Event.SourceId);
		
(* Event status ******************************************************)
	NoOfActiveEvents										:= Event.NoOfActiveEvents + SEL(EventDiagMessage.Status.31 , 0, 1);
 	EventStatus												:= Event.Status OR EventDiagMessage.Status;

		
(* Set events at the end to allow set to false in inherited FBs ********************)
	Event.no[1].Flag 										:= NOT Status.ReadyToSwitchOn; 
	Event.no[2].Flag 										:= Status.Fault;
	Event.no[3].Flag 										:= Status.Warning; 				
	Event.no[4].Flag 										:= Status.InternalLimitActive AND NOT Options.0;
	Event.no[5].Flag 										:= Status.SwitchOnDisabled;
//	Event.no[6].Flag 										:= NOT Status.FollowCmdValue AND Status.SwitchedOn AND NOT options.1 AND NOT rAxis.Status.OpMode.SimulationAxis;
	Event.no[7].Flag 										:= BrakeUnlock OR BrakeUnlocked; 	
	Event.no[8].Flag 										:= ErrorLimitPos;
	Event.no[9].Flag 										:= ErrorLimitNeg;
	
(************************************************************************)
	_callEvents												:= TRUE;
(******************************************************************************)
END_METHOD

METHOD PUBLIC confirm : bool
VAR_INPUT
END_VAR
confirm 								:= Event.confirm();
END_METHOD

PROPERTY PUBLIC optDisabledRemoteCntrNotActive : BOOL
GET
optDisabledRemoteCntrNotActive := Options.1;
END_GET
SET
Options.1 := optDisabledRemoteCntrNotActive;
END_SET
END_PROPERTY

PROPERTY PUBLIC optDisableIntLimitWarning : BOOL
GET
optDisableIntLimitWarning := Options.0;
END_GET
SET
Options.0 := optDisableIntLimitWarning;
END_SET
END_PROPERTY

END_FUNCTION_BLOCK

// POUs/IO/Drives/CoE/CiA_DS402Controlword
FUNCTION_BLOCK CiA_DS402Controlword
VAR_INPUT
	SwitchOn 				: BOOL;	// BIT 0 
	EnableVoltage 			: BOOL := TRUE; // Bit 1  
	QuickStopOK 			: BOOL := TRUE; // Bit 2 inverse signal / TRUE = RUN -
	EnableOperation 		: BOOL; // Bit 3 
//	Operation mode specific Bit 4 	: BOOL; // Bit 4
//	Operation mode specific Bit 5 	: BOOL; // Bit 5
//	Operation mode specific Bit 6 	: BOOL; // Bit 6
	FaultReset 				: BOOL; // Bit 7 
	Halt 					: BOOL; // Bit 8 - Pauses the drive in all modes
//	Operation mode specific Bit 9 	: BOOL; // Bit 9 - 
//	Reserved Bit 10 	: BOOL; // Bit 10
//	Manufacturere specific Bit 11 	: BOOL; // Bit 11
//	Manufacturere specific Bit 12 	: BOOL; // Bit 12
//	Manufacturere specific Bit 13 	: BOOL; // Bit 13
//	Manufacturere specific Bit 14 	: BOOL; // Bit 14
//	Manufacturere specific Bit 15 	: BOOL; // Bit 15	
END_VAR
VAR_OUTPUT
	Cmd						:	eCiA_DS402_CONTROL_CMD;
END_VAR
VAR
END_VAR

;

METHOD PUBLIC createControlword : BOOL
VAR_INPUT
	StatusState												: 	eCiA_DS402_STATUS_STATE;
END_VAR
VAR_IN_OUT
	Controlword												:	UINT;
END_VAR
(* work local state machine for control ****************************************************)
	CASE StatusState OF
	eCiA_DS402_STATUS_STATE.NOT_READY_TO_SWITCH_ON:
		Controlword.0										:= FALSE;
		Controlword.1										:= FALSE;
		Controlword.2										:= FALSE;
		Controlword.3										:= FALSE;
		Cmd													:= eCiA_DS402_CONTROL_CMD.DISABLE_VOLTAGE;
		
	eCiA_DS402_STATUS_STATE.SWITCH_ON_DISABLED:
		IF EnableVoltage
		THEN //back to "not ready to switch on"
			Controlword.0									:= FALSE;
			Controlword.1									:= TRUE;
			Controlword.2									:= TRUE;
			Controlword.3									:= FALSE;
			Cmd												:= eCiA_DS402_CONTROL_CMD.SHUTDOWN;
		ELSE //To "Ready to switch on"
			Controlword.0									:= FALSE;
			Controlword.1									:= FALSE;
			Controlword.2									:= FALSE;
			Controlword.3									:= FALSE;
			Cmd												:= eCiA_DS402_CONTROL_CMD.DISABLE_VOLTAGE;
		END_IF
		
	eCiA_DS402_STATUS_STATE.READY_TO_SWITCH_ON:
		IF NOT EnableVoltage
		THEN //Back to switched on disabled
			Controlword.0									:= FALSE;
			Controlword.1									:= FALSE;
			Controlword.2									:= FALSE;
			Controlword.3									:= FALSE;
			Cmd												:= eCiA_DS402_CONTROL_CMD.DISABLE_VOLTAGE;
		ELSIF SwitchOn
		THEN //To switched on
			Controlword.0									:= TRUE;
			Controlword.1									:= TRUE;
			Controlword.2									:= QuickStopOK;
			Controlword.3									:= FALSE;
			Cmd												:= eCiA_DS402_CONTROL_CMD.SWITCH_ON;	
		ELSE
			Controlword.0									:= FALSE;
			Controlword.1									:= TRUE;
			Controlword.2									:= QuickStopOK;
			Controlword.3									:= FALSE;
			Cmd												:= eCiA_DS402_CONTROL_CMD.SHUTDOWN;			
		END_IF	
		
	eCiA_DS402_STATUS_STATE.SWITCHED_ON:
		IF NOT EnableVoltage
		THEN //Back to switched on disabled
			Controlword.0									:= FALSE;
			Controlword.1									:= FALSE;
			Controlword.2									:= FALSE;
			Controlword.3									:= FALSE;
			Cmd												:= eCiA_DS402_CONTROL_CMD.DISABLE_VOLTAGE;
		ELSIF NOT SwitchOn
		THEN
			Controlword.0									:= FALSE;
			Controlword.1									:= TRUE;
			Controlword.2									:= QuickStopOK;
			Controlword.3									:= FALSE;
			Cmd												:= eCiA_DS402_CONTROL_CMD.SHUTDOWN;

		ELSIF EnableOperation
		THEN // To operation enabled
			Controlword.0									:= TRUE;
			Controlword.1									:= TRUE;
			Controlword.2									:= QuickStopOK;
			Controlword.3									:= TRUE;
			Cmd												:= SEL(QuickStopOK,eCiA_DS402_CONTROL_CMD.QUICK_STOP,eCiA_DS402_CONTROL_CMD.ENABLE_OPERATION);												
		ELSE
			Controlword.0									:= TRUE;
			Controlword.1									:= TRUE;
			Controlword.2									:= QuickStopOK;
			Controlword.3									:= FALSE;
			Cmd												:= eCiA_DS402_CONTROL_CMD.SWITCH_ON;						
		END_IF
		
	eCiA_DS402_STATUS_STATE.OPERATION_ENABLED:
		IF NOT EnableVoltage
		THEN //Back to switch on disabled
			Controlword.0									:= FALSE;
			Controlword.1									:= FALSE;
			Controlword.2									:= FALSE;
			Controlword.3									:= FALSE;
			Cmd												:= eCiA_DS402_CONTROL_CMD.DISABLE_VOLTAGE;
		ELSIF NOT SwitchOn		
		THEN // back to ready to switch on 
			Controlword.0									:= FALSE;
			Controlword.1									:= TRUE;
			Controlword.2									:= QuickStopOK;
			Controlword.3									:= FALSE;
			Cmd												:= eCiA_DS402_CONTROL_CMD.SHUTDOWN;	
		ELSIF NOT EnableOperation 
		THEN //go back to switched on
			Controlword.0									:= TRUE;
			Controlword.1									:= TRUE;
			Controlword.2									:= QuickStopOK;
			Controlword.3									:= FALSE;
			Cmd												:= eCiA_DS402_CONTROL_CMD.SWITCH_ON;
		ELSE
			Controlword.0									:= TRUE;
			Controlword.1									:= TRUE;
			Controlword.2									:= QuickStopOK;
			Controlword.3									:= TRUE;
			Cmd												:= SEL(QuickStopOK,eCiA_DS402_CONTROL_CMD.QUICK_STOP,eCiA_DS402_CONTROL_CMD.ENABLE_OPERATION);												
		END_IF
		
	eCiA_DS402_STATUS_STATE.QUICK_STOP_ACTIVE:
		IF NOT EnableVoltage
		THEN //Back to switch on disabled
			Controlword.0									:= FALSE;
			Controlword.1									:= FALSE;
			Controlword.2									:= FALSE;
			Controlword.3									:= FALSE;
			Cmd												:= eCiA_DS402_CONTROL_CMD.DISABLE_VOLTAGE;
		ELSIF NOT SwitchOn		
		THEN // back to ready to switch on 
			Controlword.0									:= FALSE;
			Controlword.1									:= TRUE;
			Controlword.2									:= QuickStopOK;
			Controlword.3									:= FALSE;
			Cmd												:= eCiA_DS402_CONTROL_CMD.SHUTDOWN;		
		ELSIF NOT EnableOperation 
		THEN //go back to switched on
			Controlword.0									:= TRUE;
			Controlword.1									:= TRUE;
			Controlword.2									:= QuickStopOK;
			Controlword.3									:= FALSE;
			Cmd												:= eCiA_DS402_CONTROL_CMD.SWITCH_ON;
		ELSE
			Controlword.0									:= TRUE;
			Controlword.1									:= TRUE;
			Controlword.2									:= QuickStopOK;
			Controlword.3									:= TRUE;
			Cmd												:= SEL(QuickStopOK,eCiA_DS402_CONTROL_CMD.QUICK_STOP,eCiA_DS402_CONTROL_CMD.ENABLE_OPERATION);												
		END_IF
		
	eCiA_DS402_STATUS_STATE.FAULT_ACTIVE:
		IF NOT EnableVoltage
		THEN //back to "not ready to switch on"
			Controlword.0									:= FALSE;
			Controlword.1									:= FALSE;
			Controlword.2									:= FALSE;
			Controlword.3									:= FALSE;
			Cmd												:= eCiA_DS402_CONTROL_CMD.DISABLE_VOLTAGE;
		ELSE //To "Ready to switch on"
			Controlword.0									:= FALSE;
			Controlword.1									:= TRUE;
			Controlword.2									:= QuickStopOK;
			Controlword.3									:= FALSE;
			Cmd												:= eCiA_DS402_CONTROL_CMD.SHUTDOWN;	
		END_IF
		
	eCiA_DS402_STATUS_STATE.FAULT_REACTION_ACTIVE:
		;	
	END_CASE
	
(* Write controlword ********************************************************)
	Controlword.7											:= FaultReset; 
	createControlword										:= TRUE;
(*****************************************************************************)
END_METHOD

END_FUNCTION_BLOCK

// POUs/IO/Drives/DC/Ey73xx/AxDriveDC
{attribute 'no_check'}
//Beckhoff Stepper terminal status and diagnoses/ EP Box used with NC axis
//EventHandling instance use inside
FUNCTION_BLOCK AxDriveDC EXTENDS AxDriveBase
VAR CONSTANT         	
END_VAR  
VAR_INPUT
END_VAR                     					
VAR_IN_OUT                  					
END_VAR                     					
VAR_OUTPUT                  					
	Status_ReadyToEnable									: BOOL;
	Status_Ready											: BOOL;
	Status_Warning											: BOOL;
	Status_Error											: BOOL;
	Status_MovingPos										: BOOL;
	Status_MovingNeg										: BOOL;
	Status_TorqueReduced									: BOOL;
	Status_DigInput1										: BOOL;
	Status_DigInput2										: BOOL;
	Status_SyncError										: BOOL;
	Status_TxPDOToggle										: BOOL;
	InfoData1										AT %I*	:	UINT;
	InfoData2										AT %I*	:	UINT;
END_VAR                     					                   					
VAR                         					
END_VAR
VAR

(* Cache *********************************************************************)
	StatusTrig												:	BYTE;
	MemStatusTrig											:	BYTE;
	MemCoeCache												: 	ARRAY[0..5] OF BYTE; //Index A020/A030 with a lenght of 17 subindex	
	
//Diag read by CoE
	Diag_Saturated											: BOOL; // Driver stage operates with maximum duty cycle
	Diag_OverTemperature 									: BOOL; // Internal terminal temperature is higher than 80°C (see subindex 0xF80F:04)
	Diag_TorqueOverloaded 									: BOOL; // Motor current is higher than the rated current
	Diag_UnderVoltage 										: BOOL; // Motor supply voltage is 20% lower than the configured nominal voltage
	Diag_OverVoltage 										: BOOL; // Motor supply voltage is 10% higher than the configured nominal voltage
	Diag_ShortCircuit 										: BOOL; // Short circuit 
	Diag_ShortCircuitB										: BOOL; // Short circuit
	Diag_NoControlPower 									: BOOL; // Control voltage at the power contacts is less than 12 V
	Diag_MiscError 											: BOOL; // Terminal initialization failed, or supply voltage is less than 8 V, or internal terminal temperature is higher than 100°C (see subindex 0xF80F:05)
	Diag_Configuration 										: BOOL; // CoE change has not yet been adopted into the current configuration
	Diag_MotorStall											: BOOL; // A loss of step has occurred
	Diag_OpenLoadA											: BOOL; // Open load on coil A - e.g. no motor connected
	Diag_OpenLoadB											: BOOL; // Open load on coil B - e.g. no motor connected

	Diag_ActualMode											: BYTE; // Current operating mode (relevant for activated automatic mode, see 0x8012:01)
	
